C03654=1154.886,184.400,-60.410,-178.214,7.081,148.800
C03655=1154.890,184.131,-60.386,-178.217,7.080,148.800
C03656=1154.895,183.861,-60.360,-178.220,7.077,148.801
C03657=1154.900,183.591,-60.335,-178.223,7.075,148.801
C03658=1154.905,183.322,-60.310,-178.226,7.073,148.801
C03659=1154.909,183.073,-60.287,-178.229,7.070,148.801
C03660=1154.915,182.824,-60.264,-178.231,7.068,148.802
C03661=1154.919,182.576,-60.241,-178.234,7.066,148.802
C03662=1154.924,182.326,-60.218,-178.237,7.063,148.802
C03663=1154.928,182.077,-60.195,-178.240,7.062,148.803
C03664=1154.932,181.828,-60.172,-178.242,7.060,148.803
C03665=1154.938,181.580,-60.149,-178.245,7.057,148.803
C03666=1154.942,181.331,-60.126,-178.248,7.055,148.804
C03667=1154.946,181.082,-60.103,-178.251,7.053,148.804
C03668=1154.951,180.832,-60.080,-178.254,7.051,148.804
C03669=1154.956,180.583,-60.057,-178.256,7.049,148.804
C03670=1154.961,180.335,-60.035,-178.259,7.046,148.805
C03671=1154.965,180.086,-60.011,-178.262,7.045,148.805
C03672=1154.970,179.837,-59.989,-178.264,7.043,148.805
C03673=1154.974,179.588,-59.966,-178.267,7.040,148.806
C03674=1154.979,179.339,-59.943,-178.270,7.038,148.806
C03675=1154.984,179.091,-59.920,-178.272,7.036,148.806
C03676=1154.989,178.841,-59.898,-178.276,7.034,148.806
C03677=1154.993,178.593,-59.875,-178.278,7.032,148.807
C03678=1154.997,178.343,-59.851,-178.281,7.030,148.807
C03679=1155.002,178.095,-59.830,-178.284,7.027,148.807
C03680=1155.007,177.846,-59.806,-178.286,7.025,148.808
C03681=1155.012,177.596,-59.784,-178.289,7.024,148.808
C03682=1155.016,177.348,-59.761,-178.292,7.021,148.808
C03683=1155.021,177.099,-59.738,-178.295,7.019,148.808
C03684=1155.025,176.850,-59.716,-178.297,7.017,148.809
C03685=1155.030,176.601,-59.693,-178.301,7.015,148.809
C03686=1155.035,176.352,-59.671,-178.303,7.013,148.809
C03687=1155.040,176.103,-59.648,-178.306,7.011,148.810
C03688=1155.044,175.854,-59.625,-178.309,7.008,148.810
C03689=1155.048,175.606,-59.603,-178.311,7.007,148.810
C03690=1155.053,175.357,-59.580,-178.314,7.004,148.811
C03691=1155.057,175.107,-59.558,-178.317,7.002,148.811
C03692=1155.063,174.859,-59.535,-178.320,7.000,148.811
C03693=1155.067,174.610,-59.513,-178.322,6.998,148.812
C03694=1155.072,174.361,-59.489,-178.325,6.996,148.812
C03695=1155.077,174.112,-59.468,-178.328,6.994,148.812
C03696=1155.082,173.862,-59.445,-178.331,6.992,148.812
C03697=1155.086,173.614,-59.422,-178.334,6.989,148.813
C03698=1155.090,173.365,-59.401,-178.336,6.987,148.813
C03699=1155.095,173.116,-59.377,-178.339,6.986,148.813
C03700=1155.099,172.867,-59.355,-178.341,6.984,148.814
C03701=1155.104,172.619,-59.333,-178.345,6.981,148.814
C03702=1155.109,172.369,-59.310,-178.347,6.979,148.814
C03703=1155.114,172.120,-59.288,-178.350,6.977,148.815
C03704=1155.118,171.871,-59.265,-178.353,6.975,148.815
C03705=1155.123,171.622,-59.243,-178.356,6.973,148.815
C03706=1155.128,171.373,-59.221,-178.358,6.971,148.815
C03707=1155.132,171.124,-59.198,-178.361,6.969,148.816
C03708=1155.137,170.876,-59.176,-178.364,6.967,148.816
C03709=1155.141,170.626,-59.154,-178.366,6.965,148.817
C03710=1155.145,170.378,-59.131,-178.369,6.963,148.817
C03711=1155.151,170.129,-59.109,-178.372,6.960,148.817
C03712=1155.155,169.879,-59.087,-178.375,6.959,148.817
C03713=1155.160,169.631,-59.065,-178.377,6.957,148.818
C03714=1155.165,169.382,-59.042,-178.380,6.955,148.818
C03715=1155.170,169.133,-59.020,-178.383,6.953,148.818
C03716=1155.174,168.884,-58.998,-178.386,6.951,148.819
C03717=1155.179,168.635,-58.977,-178.388,6.949,148.819
C03718=1155.184,168.385,-58.954,-178.392,6.946,148.819
C03719=1155.188,168.137,-58.932,-178.394,6.945,148.820
C03720=1155.193,167.888,-58.910,-178.397,6.943,148.820
C03721=1155.197,167.639,-58.888,-178.399,6.941,148.820
C03722=1155.203,167.390,-58.865,-178.402,6.938,148.821
C03723=1155.207,167.140,-58.843,-178.405,6.936,148.821
C03724=1155.212,166.892,-58.822,-178.408,6.935,148.821
C03725=1155.216,166.642,-58.799,-178.411,6.933,148.822
C03726=1155.221,166.394,-58.778,-178.413,6.930,148.822
C03727=1155.225,166.145,-58.755,-178.416,6.928,148.822
C03728=1155.230,165.896,-58.733,-178.419,6.927,148.823
C03729=1155.235,165.647,-58.711,-178.421,6.925,148.823
C03730=1155.240,165.398,-58.689,-178.425,6.922,148.823
C03731=1155.244,165.149,-58.667,-178.427,6.920,148.823
C03732=1155.249,164.900,-58.645,-178.430,6.918,148.824
C03733=1155.254,164.651,-58.624,-178.432,6.917,148.824
C03734=1155.258,164.402,-58.602,-178.436,6.914,148.825
C03735=1155.263,164.153,-58.580,-178.438,6.912,148.825
C03736=1155.268,163.904,-58.557,-178.441,6.911,148.825
C03737=1155.273,163.655,-58.536,-178.443,6.909,148.825
C03738=1155.277,163.406,-58.513,-178.446,6.906,148.826
C03739=1155.282,163.157,-58.492,-178.449,6.904,148.826
C03740=1155.286,162.908,-58.470,-178.452,6.903,148.827
C03741=1155.291,162.659,-58.448,-178.455,6.901,148.827
C03742=1155.296,162.410,-58.427,-178.457,6.899,148.827
C03743=1155.300,162.161,-58.405,-178.461,6.897,148.828
C03744=1155.305,161.912,-58.383,-178.463,6.894,148.828
C03745=1155.309,161.663,-58.361,-178.465,6.893,148.828
C03746=1155.314,161.414,-58.340,-178.468,6.891,148.829
C03747=1155.319,161.165,-58.318,-178.471,6.888,148.829
C03748=1155.323,160.916,-58.296,-178.474,6.887,148.829
C03749=1155.328,160.667,-58.274,-178.477,6.885,148.830
C03750=1155.333,160.417,-58.253,-178.480,6.883,148.830
C03751=1155.338,160.169,-58.231,-178.482,6.881,148.830
C03752=1155.343,159.920,-58.210,-178.485,6.879,148.831
C03753=1155.347,159.671,-58.187,-178.488,6.877,148.831
C03754=1155.352,159.421,-58.167,-178.490,6.875,148.831
C03755=1155.357,159.173,-58.145,-178.493,6.873,148.832
C03756=1155.361,158.924,-58.123,-178.496,6.872,148.832
C03757=1155.366,158.675,-58.101,-178.499,6.869,148.832
C03758=1155.371,158.426,-58.080,-178.501,6.867,148.833
C03759=1155.376,158.157,-58.057,-178.504,6.865,148.833
C03760=1155.381,157.888,-58.033,-178.508,6.863,148.834
C03761=1155.386,157.619,-58.011,-178.511,6.861,148.834
C03762=1155.391,157.350,-57.986,-178.514,6.859,148.834
C03763=1155.396,157.101,-57.966,-178.516,6.857,148.834
C03764=1155.400,156.852,-57.944,-178.519,6.855,148.835
C03765=1155.405,156.603,-57.922,-178.521,6.853,148.835
C03766=1155.410,156.354,-57.901,-178.524,6.851,148.836
C03767=1155.414,156.105,-57.879,-178.527,6.850,148.836
C03768=1155.419,155.855,-57.858,-178.530,6.847,148.836
C03769=1155.424,155.607,-57.837,-178.533,6.845,148.837
C03770=1155.428,155.358,-57.815,-178.536,6.844,148.837
C03771=1155.433,155.108,-57.794,-178.538,6.842,148.837
C03772=1155.438,154.860,-57.773,-178.541,6.840,148.838
C03773=1155.443,154.610,-57.752,-178.543,6.838,148.838
C03774=1155.447,154.361,-57.730,-178.546,6.836,148.838
C03775=1155.452,154.112,-57.709,-178.549,6.834,148.839
C03776=1155.456,153.863,-57.688,-178.552,6.832,148.839
C03777=1155.462,153.614,-57.667,-178.555,6.830,148.839
C03778=1155.466,153.365,-57.645,-178.557,6.829,148.840
C03779=1155.471,153.116,-57.624,-178.560,6.827,148.840
C03780=1155.475,152.867,-57.602,-178.563,6.824,148.841
C03781=1155.480,152.618,-57.582,-178.566,6.823,148.841
C03782=1155.485,152.369,-57.560,-178.569,6.821,148.841
C03783=1155.490,152.119,-57.538,-178.571,6.819,148.842
C03784=1155.494,151.871,-57.517,-178.574,6.817,148.842
C03785=1155.499,151.622,-57.496,-178.576,6.815,148.842
C03786=1155.504,151.373,-57.475,-178.579,6.814,148.843
C03787=1155.508,151.124,-57.454,-178.582,6.811,148.843
C03788=1155.513,150.874,-57.433,-178.585,6.809,148.843
C03789=1155.518,150.625,-57.412,-178.588,6.808,148.844
C03790=1155.522,150.377,-57.391,-178.590,6.806,148.844
C03791=1155.528,150.127,-57.370,-178.593,6.804,148.845
C03792=1155.533,149.878,-57.349,-178.596,6.803,148.845
C03793=1155.537,149.630,-57.328,-178.598,6.801,148.845
C03794=1155.541,149.380,-57.307,-178.601,6.799,148.846
C03795=1155.547,149.131,-57.286,-178.604,6.797,148.846
C03796=1155.551,148.882,-57.265,-178.607,6.795,148.846
C03797=1155.556,148.633,-57.244,-178.610,6.793,148.847
C03798=1155.561,148.384,-57.223,-178.613,6.791,148.847
C03799=1155.565,148.135,-57.202,-178.615,6.790,148.848
C03800=1155.570,147.886,-57.181,-178.618,6.788,148.848
C03801=1155.574,147.637,-57.160,-178.620,6.786,148.848
C03802=1155.579,147.387,-57.139,-178.623,6.784,148.849
C03803=1155.585,147.138,-57.118,-178.626,6.782,148.849
C03804=1155.589,146.890,-57.097,-178.629,6.780,148.849
C03805=1155.594,146.640,-57.076,-178.632,6.778,148.850
C03806=1155.598,146.391,-57.055,-178.634,6.776,148.850
C03807=1155.603,146.142,-57.035,-178.637,6.775,148.850
C03808=1155.608,145.893,-57.014,-178.640,6.773,148.851
C03809=1155.613,145.644,-56.993,-178.642,6.771,148.851
C03810=1155.618,145.395,-56.973,-178.645,6.769,148.852
C03811=1155.622,145.146,-56.951,-178.648,6.768,148.852
C03812=1155.626,144.897,-56.930,-178.651,6.766,148.852
C03813=1155.631,144.648,-56.909,-178.653,6.764,148.853
C03814=1155.636,144.399,-56.889,-178.657,6.762,148.853
C03815=1155.641,144.149,-56.868,-178.659,6.760,148.853
C03816=1155.645,143.900,-56.848,-178.662,6.758,148.854
C03817=1155.651,143.651,-56.827,-178.665,6.757,148.854
C03818=1155.655,143.402,-56.806,-178.667,6.755,148.855
C03819=1155.660,143.153,-56.785,-178.670,6.753,148.855
C03820=1155.665,142.904,-56.765,-178.673,6.751,148.855
C03821=1155.669,142.655,-56.745,-178.676,6.750,148.856
C03822=1155.674,142.406,-56.724,-178.678,6.748,148.856
C03823=1155.679,142.157,-56.703,-178.681,6.746,148.857
C03824=1155.684,141.908,-56.682,-178.684,6.745,148.857
C03825=1155.688,141.659,-56.662,-178.686,6.743,148.857
C03826=1155.694,141.409,-56.641,-178.689,6.741,148.858
C03827=1155.698,141.160,-56.621,-178.692,6.739,148.858
C03828=1155.702,140.911,-56.600,-178.695,6.737,148.859
C03829=1155.708,140.662,-56.579,-178.698,6.735,148.859
C03830=1155.712,140.413,-56.559,-178.700,6.733,148.859
C03831=1155.716,140.164,-56.539,-178.703,6.732,148.860
C03832=1155.722,139.914,-56.518,-178.706,6.730,148.860
C03833=1155.726,139.665,-56.498,-178.709,6.728,148.860
C03834=1155.731,139.416,-56.478,-178.711,6.726,148.861
C03835=1155.736,139.167,-56.457,-178.714,6.725,148.861
C03836=1155.740,138.918,-56.436,-178.717,6.723,148.862
C03837=1155.745,138.669,-56.416,-178.719,6.721,148.862
C03838=1155.750,138.419,-56.396,-178.722,6.720,148.862
C03839=1155.755,138.171,-56.375,-178.725,6.718,148.863
C03840=1155.759,137.922,-56.355,-178.728,6.716,148.863
C03841=1155.764,137.672,-56.334,-178.730,6.714,148.864
C03842=1155.769,137.423,-56.314,-178.733,6.713,148.864
C03843=1155.774,137.174,-56.294,-178.736,6.711,148.864
C03844=1155.779,136.926,-56.274,-178.738,6.709,148.865
C03845=1155.784,136.676,-56.253,-178.741,6.708,148.865
C03846=1155.788,136.427,-56.233,-178.744,6.706,148.866
C03847=1155.793,136.178,-56.213,-178.747,6.704,148.866
C03848=1155.797,135.929,-56.193,-178.749,6.702,148.866
C03849=1155.803,135.680,-56.172,-178.752,6.701,148.867
C03850=1155.807,135.430,-56.152,-178.755,6.699,148.867
C03851=1155.812,135.181,-56.132,-178.757,6.697,148.867
C03852=1155.816,134.932,-56.111,-178.761,6.695,148.868
C03853=1155.822,134.683,-56.092,-178.764,6.693,148.868
C03854=1155.827,134.434,-56.071,-178.767,6.692,148.869
C03855=1155.831,134.185,-56.051,-178.769,6.690,148.869
C03856=1155.836,133.935,-56.031,-178.772,6.688,148.870
C03857=1155.840,133.686,-56.010,-178.775,6.686,148.870
C03858=1155.845,133.437,-55.991,-178.777,6.685,148.870
C03859=1155.849,133.188,-55.970,-178.780,6.683,148.871
C03860=1155.855,132.939,-55.951,-178.783,6.681,148.871
C03861=1155.860,132.690,-55.930,-178.786,6.680,148.872
C03862=1155.864,132.441,-55.910,-178.788,6.678,148.872
C03863=1155.869,132.172,-55.889,-178.791,6.676,148.872
C03864=1155.875,131.903,-55.867,-178.794,6.674,148.873
C03865=1155.880,131.635,-55.845,-178.797,6.673,148.873
C03866=1155.885,131.366,-55.824,-178.800,6.671,148.874
C03867=1155.890,131.117,-55.804,-178.802,6.670,148.874
C03868=1155.894,130.868,-55.784,-178.805,6.668,148.875
C03869=1155.900,130.619,-55.764,-178.808,6.666,148.875
C03870=1155.904,130.370,-55.744,-178.810,6.664,148.875
C03871=1155.909,130.120,-55.724,-178.813,6.663,148.876
C03872=1155.913,129.871,-55.704,-178.816,6.661,148.876
C03873=1155.919,129.623,-55.685,-178.819,6.659,148.877
C03874=1155.923,129.373,-55.665,-178.821,6.658,148.877
C03875=1155.928,129.124,-55.645,-178.824,6.656,148.878
C03876=1155.933,128.874,-55.625,-178.827,6.655,148.878
C03877=1155.938,128.626,-55.605,-178.830,6.653,148.878
C03878=1155.942,128.377,-55.585,-178.833,6.651,148.879
C03879=1155.947,128.127,-55.566,-178.835,6.649,148.879
C03880=1155.952,127.878,-55.545,-178.838,6.648,148.880
C03881=1155.957,127.629,-55.526,-178.841,6.646,148.880
C03882=1155.962,127.380,-55.506,-178.843,6.644,148.880
C03883=1155.966,127.131,-55.486,-178.846,6.643,148.881
C03884=1155.971,126.881,-55.466,-178.849,6.641,148.881
C03885=1155.976,126.632,-55.447,-178.852,6.639,148.882
C03886=1155.981,126.383,-55.427,-178.855,6.638,148.882
C03887=1155.985,126.134,-55.407,-178.858,6.636,148.883
C03888=1155.991,125.885,-55.388,-178.860,6.634,148.883
C03889=1155.996,125.635,-55.368,-178.863,6.633,148.883
C03890=1155.999,125.387,-55.348,-178.866,6.631,148.884
C03891=1156.004,125.137,-55.329,-178.868,6.629,148.884
C03892=1156.009,124.888,-55.309,-178.871,6.627,148.885
C03893=1156.014,124.639,-55.290,-178.874,6.626,148.885
C03894=1156.019,124.389,-55.270,-178.876,6.625,148.885
C03895=1156.024,124.141,-55.250,-178.879,6.623,148.886
C03896=1156.029,123.891,-55.230,-178.882,6.622,148.886
C03897=1156.033,123.642,-55.211,-178.885,6.620,148.887
C03898=1156.038,123.393,-55.192,-178.887,6.618,148.887
C03899=1156.043,123.144,-55.172,-178.890,6.617,148.888
C03900=1156.047,122.894,-55.153,-178.893,6.615,148.888
C03901=1156.053,122.645,-55.133,-178.895,6.613,148.888
C03902=1156.057,122.396,-55.114,-178.898,6.612,148.889
C03903=1156.063,122.147,-55.094,-178.901,6.610,148.889
C03904=1156.067,121.898,-55.075,-178.904,6.608,148.890
C03905=1156.071,121.649,-55.055,-178.907,6.607,148.890
C03906=1156.077,121.400,-55.036,-178.909,6.605,148.891
C03907=1156.081,121.150,-55.016,-178.912,6.603,148.891
C03908=1156.086,120.901,-54.996,-178.914,6.602,148.891
C03909=1156.091,120.652,-54.978,-178.917,6.601,148.892
C03910=1156.095,120.402,-54.958,-178.920,6.599,148.892
C03911=1156.101,120.154,-54.939,-178.922,6.597,148.893
C03912=1156.106,119.904,-54.919,-178.926,6.596,148.893
C03913=1156.110,119.655,-54.900,-178.928,6.594,148.894
C03914=1156.115,119.406,-54.881,-178.931,6.593,148.894
C03915=1156.120,119.156,-54.861,-178.934,6.591,148.894
C03916=1156.125,118.907,-54.842,-178.937,6.589,148.895
C03917=1156.129,118.658,-54.823,-178.939,6.587,148.895
C03918=1156.134,118.409,-54.803,-178.941,6.587,148.896
C03919=1156.139,118.160,-54.784,-178.945,6.585,148.896
C03920=1156.144,117.911,-54.766,-178.947,6.583,148.897
C03921=1156.149,117.661,-54.746,-178.950,6.582,148.897
C03922=1156.154,117.412,-54.727,-178.953,6.580,148.897
C03923=1156.158,117.163,-54.708,-178.955,6.578,148.898
C03924=1156.163,116.913,-54.688,-178.958,6.577,148.898
C03925=1156.168,116.664,-54.669,-178.961,6.575,148.899
C03926=1156.172,116.415,-54.650,-178.964,6.574,148.899
C03927=1156.178,116.166,-54.630,-178.966,6.573,148.900
C03928=1156.183,115.916,-54.611,-178.969,6.571,148.900
C03929=1156.187,115.668,-54.593,-178.972,6.569,148.901
C03930=1156.192,115.418,-54.573,-178.974,6.568,148.901
C03931=1156.197,115.169,-54.554,-178.977,6.566,148.901
C03932=1156.201,114.920,-54.535,-178.980,6.565,148.902
C03933=1156.207,114.670,-54.516,-178.983,6.563,148.902
C03934=1156.211,114.421,-54.497,-178.986,6.561,148.903
C03935=1156.216,114.172,-54.478,-178.988,6.560,148.903
C03936=1156.221,113.924,-54.459,-178.991,6.558,148.904
C03937=1156.226,113.674,-54.440,-178.993,6.557,148.904
C03938=1156.231,113.425,-54.421,-178.997,6.555,148.905
C03939=1156.235,113.175,-54.402,-178.999,6.554,148.905
C03940=1156.241,112.926,-54.383,-179.002,6.552,148.905
C03941=1156.245,112.677,-54.364,-179.005,6.550,148.906
C03942=1156.250,112.428,-54.345,-179.007,6.549,148.906
C03943=1156.255,112.178,-54.327,-179.010,6.548,148.907
C03944=1156.260,111.929,-54.307,-179.013,6.546,148.907
C03945=1156.265,111.681,-54.289,-179.015,6.545,148.908
C03946=1156.270,111.430,-54.270,-179.018,6.543,148.908
C03947=1156.274,111.182,-54.251,-179.021,6.541,148.909
C03948=1156.279,110.932,-54.232,-179.024,6.540,148.909
C03949=1156.284,110.683,-54.213,-179.026,6.539,148.910
C03950=1156.289,110.433,-54.194,-179.029,6.537,148.910
C03951=1156.293,110.184,-54.176,-179.032,6.536,148.910
C03952=1156.299,109.935,-54.156,-179.034,6.534,148.911
C03953=1156.303,109.686,-54.138,-179.037,6.532,148.911
C03954=1156.308,109.437,-54.119,-179.040,6.531,148.912
C03955=1156.313,109.188,-54.101,-179.042,6.530,148.912
C03956=1156.317,108.938,-54.082,-179.045,6.528,148.913
C03957=1156.323,108.689,-54.063,-179.048,6.527,148.913
C03958=1156.327,108.440,-54.044,-179.051,6.525,148.913
C03959=1156.333,108.190,-54.026,-179.054,6.524,148.914
C03960=1156.337,107.941,-54.007,-179.056,6.523,148.915
C03961=1156.342,107.691,-53.988,-179.059,6.521,148.915
C03962=1156.347,107.443,-53.969,-179.061,6.519,148.915
C03963=1156.352,107.194,-53.951,-179.064,6.518,148.916
C03964=1156.357,106.944,-53.932,-179.067,6.516,148.916
C03965=1156.362,106.695,-53.914,-179.070,6.515,148.917
C03966=1156.366,106.446,-53.895,-179.072,6.514,148.917
C03967=1156.371,106.177,-53.875,-179.075,6.512,148.918
C03968=1156.376,105.909,-53.855,-179.078,6.511,148.918
C03969=1156.382,105.641,-53.834,-179.081,6.509,148.919
C03970=1156.387,105.373,-53.815,-179.084,6.508,148.919
C03971=1156.392,105.122,-53.796,-179.087,6.506,148.920
C03972=1156.397,104.874,-53.777,-179.090,6.504,148.920
C03973=1156.402,104.625,-53.759,-179.092,6.502,148.921
C03974=1156.407,104.374,-53.740,-179.095,6.501,148.921
C03975=1156.412,104.125,-53.722,-179.098,6.500,148.922
C03976=1156.416,103.877,-53.704,-179.100,6.499,148.922
C03977=1156.421,103.628,-53.686,-179.103,6.497,148.922
C03978=1156.426,103.377,-53.667,-179.106,6.495,148.923
C03979=1156.431,103.129,-53.648,-179.109,6.494,148.923
C03980=1156.436,102.880,-53.630,-179.111,6.493,148.924
C03981=1156.441,102.630,-53.612,-179.114,6.491,148.924
C03982=1156.446,102.380,-53.593,-179.117,6.490,148.925
C03983=1156.450,102.132,-53.575,-179.120,6.488,148.925
C03984=1156.455,101.882,-53.557,-179.122,6.487,148.926
C03985=1156.460,101.633,-53.539,-179.125,6.486,148.926
C03986=1156.465,101.383,-53.520,-179.127,6.484,148.927
C03987=1156.470,101.135,-53.501,-179.131,6.483,148.927
C03988=1156.475,100.885,-53.483,-179.133,6.481,148.928
C03989=1156.480,100.636,-53.465,-179.135,6.480,148.928
C03990=1156.484,100.386,-53.447,-179.138,6.478,148.928
C03991=1156.489,100.137,-53.428,-179.141,6.477,148.929
C03992=1156.494,99.888,-53.410,-179.144,6.475,148.929
C03993=1156.499,99.639,-53.392,-179.146,6.474,148.930
C03994=1156.504,99.390,-53.373,-179.149,6.473,148.930
C03995=1156.508,99.140,-53.355,-179.152,6.471,148.931
C03996=1156.513,98.891,-53.337,-179.155,6.470,148.931
C03997=1156.518,98.642,-53.319,-179.157,6.469,148.932
C03998=1156.524,98.392,-53.301,-179.160,6.467,148.932
C03999=1156.529,98.143,-53.283,-179.163,6.466,148.933
C04000=1156.534,97.894,-53.265,-179.166,6.464,148.933
C04001=1156.538,97.644,-53.246,-179.168,6.463,148.934
C04002=1156.543,97.395,-53.228,-179.171,6.461,148.934
C04003=1156.548,97.146,-53.210,-179.174,6.460,148.935
C04004=1156.553,96.896,-53.192,-179.176,6.458,148.935
C04005=1156.557,96.647,-53.174,-179.179,6.458,148.936
C04006=1156.562,96.398,-53.156,-179.181,6.456,148.936
C04007=1156.567,96.148,-53.138,-179.185,6.455,148.937
C04008=1156.572,95.899,-53.120,-179.187,6.453,148.937
C04009=1156.577,95.650,-53.102,-179.189,6.452,148.937
C04010=1156.581,95.401,-53.084,-179.192,6.450,148.938
C04011=1156.586,95.152,-53.066,-179.195,6.449,148.939
C04012=1156.591,94.902,-53.048,-179.197,6.448,148.939
C04013=1156.597,94.653,-53.029,-179.200,6.446,148.939
C04014=1156.602,94.404,-53.012,-179.203,6.445,148.940
C04015=1156.607,94.155,-52.994,-179.206,6.443,148.940
C04016=1156.611,93.905,-52.975,-179.208,6.442,148.941
C04017=1156.616,93.655,-52.957,-179.211,6.441,148.941
C04018=1156.621,93.406,-52.940,-179.214,6.439,148.942
C04019=1156.625,93.157,-52.923,-179.216,6.439,148.942
C04020=1156.630,92.908,-52.905,-179.219,6.437,148.943
C04021=1156.635,92.658,-52.887,-179.222,6.436,148.943
C04022=1156.640,92.409,-52.869,-179.225,6.434,148.944
C04023=1156.645,92.160,-52.851,-179.227,6.433,148.944
C04024=1156.650,91.910,-52.833,-179.230,6.431,148.945
C04025=1156.655,91.661,-52.815,-179.233,6.430,148.945
C04026=1156.660,91.412,-52.797,-179.235,6.429,148.946
C04027=1156.665,91.163,-52.779,-179.238,6.427,148.946
C04028=1156.670,90.914,-52.761,-179.241,6.426,148.947
C04029=1156.675,90.664,-52.744,-179.244,6.424,148.947
C04030=1156.680,90.415,-52.726,-179.246,6.423,148.948
C04031=1156.685,90.165,-52.708,-179.249,6.422,148.948
C04032=1156.689,89.917,-52.691,-179.252,6.420,148.949
C04033=1156.694,89.666,-52.673,-179.254,6.420,148.949
C04034=1156.699,89.417,-52.655,-179.257,6.418,148.950
C04035=1156.704,89.168,-52.637,-179.260,6.417,148.950
C04036=1156.709,88.918,-52.620,-179.262,6.416,148.951
C04037=1156.714,88.669,-52.602,-179.265,6.414,148.951
C04038=1156.719,88.420,-52.584,-179.268,6.413,148.952
C04039=1156.723,88.170,-52.567,-179.270,6.412,148.952
C04040=1156.728,87.921,-52.549,-179.273,6.410,148.953
C04041=1156.733,87.672,-52.532,-179.276,6.408,148.953
C04042=1156.739,87.423,-52.515,-179.278,6.408,148.954
C04043=1156.744,87.174,-52.497,-179.281,6.406,148.954
C04044=1156.749,86.924,-52.479,-179.284,6.405,148.954
C04045=1156.753,86.675,-52.462,-179.287,6.404,148.955
C04046=1156.758,86.426,-52.444,-179.289,6.402,148.955
C04047=1156.763,86.176,-52.427,-179.292,6.401,148.956
C04048=1156.768,85.927,-52.409,-179.295,6.400,148.957
C04049=1156.773,85.677,-52.392,-179.297,6.398,148.957
C04050=1156.777,85.428,-52.374,-179.300,6.397,148.957
C04051=1156.783,85.178,-52.357,-179.303,6.396,148.958
C04052=1156.788,84.929,-52.339,-179.305,6.395,148.958
C04053=1156.792,84.680,-52.321,-179.308,6.393,148.959
C04054=1156.797,84.430,-52.304,-179.311,6.392,148.960
C04055=1156.802,84.181,-52.286,-179.314,6.391,148.960
C04056=1156.807,83.931,-52.269,-179.316,6.389,148.960
C04057=1156.812,83.682,-52.252,-179.319,6.388,148.961
C04058=1156.816,83.433,-52.234,-179.322,6.387,148.961
C04059=1156.822,83.184,-52.217,-179.324,6.385,148.962
C04060=1156.826,82.935,-52.200,-179.327,6.385,148.963
C04061=1156.832,82.685,-52.183,-179.330,6.383,148.963
C04062=1156.837,82.436,-52.165,-179.332,6.381,148.963
C04063=1156.841,82.186,-52.148,-179.335,6.380,148.964
C04064=1156.846,81.937,-52.130,-179.338,6.379,148.964
C04065=1156.851,81.687,-52.113,-179.340,6.378,148.965
C04066=1156.856,81.438,-52.096,-179.343,6.376,148.965
C04067=1156.861,81.189,-52.078,-179.346,6.375,148.966
C04068=1156.866,80.940,-52.061,-179.348,6.374,148.966
C04069=1156.871,80.690,-52.045,-179.351,6.373,148.967
C04070=1156.876,80.441,-52.027,-179.354,6.371,148.967
C04071=1156.881,80.172,-52.008,-179.356,6.370,148.968
C04072=1156.886,79.904,-51.990,-179.359,6.369,148.969
C04073=1156.892,79.635,-51.971,-179.362,6.367,148.969
C04074=1156.897,79.367,-51.953,-179.365,6.366,148.970
C04075=1156.902,79.118,-51.936,-179.367,6.365,148.970
C04076=1156.907,78.869,-51.918,-179.371,6.364,148.971
C04077=1156.912,78.619,-51.902,-179.373,6.362,148.971
C04078=1156.917,78.370,-51.884,-179.376,6.361,148.972
C04079=1156.921,78.120,-51.867,-179.379,6.360,148.972
C04080=1156.927,77.871,-51.850,-179.382,6.358,148.973
C04081=1156.931,77.622,-51.834,-179.384,6.358,148.973
C04082=1156.936,77.373,-51.816,-179.387,6.356,148.974
C04083=1156.942,77.123,-51.798,-179.389,6.355,148.974
C04084=1156.946,76.873,-51.782,-179.392,6.354,148.975
C04085=1156.952,76.624,-51.765,-179.395,6.352,148.975
C04086=1156.956,76.375,-51.748,-179.397,6.351,148.976
C04087=1156.961,76.126,-51.730,-179.400,6.350,148.976
C04088=1156.966,75.876,-51.713,-179.402,6.349,148.977
C04089=1156.972,75.627,-51.697,-179.405,6.348,148.977
C04090=1156.976,75.378,-51.680,-179.408,6.347,148.978
C04091=1156.980,75.128,-51.663,-179.411,6.345,148.978
C04092=1156.986,74.878,-51.646,-179.413,6.344,148.979
C04093=1156.990,74.629,-51.629,-179.416,6.343,148.979
C04094=1156.996,74.380,-51.612,-179.419,6.342,148.980
C04095=1157.000,74.131,-51.595,-179.421,6.341,148.980
C04096=1157.005,73.881,-51.578,-179.424,6.339,148.981
C04097=1157.010,73.632,-51.561,-179.427,6.338,148.981
C04098=1157.016,73.382,-51.544,-179.429,6.337,148.982
C04099=1157.020,73.133,-51.528,-179.432,6.336,148.982
C04100=1157.025,72.883,-51.511,-179.434,6.335,148.983
C04101=1157.030,72.634,-51.494,-179.438,6.333,148.983
C04102=1157.035,72.385,-51.477,-179.440,6.332,148.984
C04103=1157.040,72.135,-51.460,-179.442,6.331,148.984
C04104=1157.045,71.886,-51.444,-179.446,6.329,148.985
C04105=1157.050,71.637,-51.427,-179.448,6.329,148.985
C04106=1157.055,71.387,-51.410,-179.451,6.327,148.986
C04107=1157.060,71.138,-51.393,-179.453,6.326,148.987
C04108=1157.064,70.889,-51.377,-179.456,6.325,148.987
C04109=1157.070,70.639,-51.360,-179.459,6.324,148.988
C04110=1157.075,70.390,-51.343,-179.461,6.323,148.988
C04111=1157.079,70.141,-51.327,-179.463,6.322,148.988
C04112=1157.084,69.891,-51.309,-179.467,6.320,148.989
C04113=1157.090,69.642,-51.293,-179.469,6.319,148.990
C04114=1157.094,69.392,-51.277,-179.472,6.318,148.990
C04115=1157.100,69.142,-51.260,-179.475,6.317,148.991
C04116=1157.105,68.893,-51.243,-179.477,6.316,148.991
C04117=1157.109,68.644,-51.227,-179.480,6.314,148.992
C04118=1157.114,68.394,-51.210,-179.482,6.314,148.992
C04119=1157.119,68.145,-51.193,-179.485,6.312,148.993
C04120=1157.124,67.896,-51.177,-179.488,6.311,148.993
C04121=1157.128,67.646,-51.160,-179.490,6.310,148.994
C04122=1157.135,67.397,-51.144,-179.493,6.309,148.994
C04123=1157.139,67.147,-51.127,-179.496,6.308,148.995
C04124=1157.144,66.898,-51.111,-179.498,6.307,148.995
C04125=1157.149,66.649,-51.094,-179.501,6.305,148.996
C04126=1157.154,66.399,-51.077,-179.504,6.304,148.996
C04127=1157.159,66.150,-51.061,-179.507,6.303,148.997
C04128=1157.164,65.900,-51.045,-179.509,6.301,148.997
C04129=1157.169,65.652,-51.028,-179.511,6.301,148.998
C04130=1157.173,65.402,-51.012,-179.515,6.299,148.999
C04131=1157.179,65.152,-50.995,-179.517,6.298,148.999
C04132=1157.184,64.903,-50.979,-179.520,6.297,149.000
C04133=1157.188,64.653,-50.962,-179.522,6.296,149.000
C04134=1157.193,64.405,-50.946,-179.525,6.295,149.000
C04135=1157.198,64.154,-50.930,-179.528,6.294,149.001
C04136=1157.203,63.906,-50.913,-179.530,6.292,149.002
C04137=1157.208,63.656,-50.896,-179.533,6.292,149.002
C04138=1157.214,63.406,-50.881,-179.536,6.290,149.003
C04139=1157.218,63.157,-50.864,-179.538,6.289,149.003
C04140=1157.223,62.908,-50.847,-179.541,6.288,149.004
C04141=1157.228,62.658,-50.832,-179.543,6.287,149.004
C04142=1157.233,62.409,-50.815,-179.546,6.286,149.005
C04143=1157.238,62.159,-50.799,-179.549,6.285,149.005
C04144=1157.243,61.909,-50.782,-179.551,6.283,149.006
C04145=1157.248,61.661,-50.766,-179.554,6.283,149.006
C04146=1157.253,61.411,-50.750,-179.557,6.281,149.007
C04147=1157.258,61.162,-50.734,-179.559,6.281,149.008
C04148=1157.263,60.912,-50.718,-179.562,6.279,149.008
C04149=1157.268,60.663,-50.701,-179.564,6.278,149.008
C04150=1157.273,60.413,-50.685,-179.567,6.277,149.009
C04151=1157.278,60.164,-50.669,-179.570,6.276,149.009
C04152=1157.282,59.915,-50.652,-179.573,6.275,149.010
C04153=1157.288,59.665,-50.637,-179.575,6.274,149.011
C04154=1157.292,59.416,-50.620,-179.578,6.273,149.011
C04155=1157.298,59.166,-50.605,-179.580,6.272,149.012
C04156=1157.302,58.917,-50.588,-179.583,6.270,149.012
C04157=1157.308,58.667,-50.572,-179.586,6.270,149.013
C04158=1157.313,58.419,-50.556,-179.588,6.268,149.013
C04159=1157.317,58.168,-50.540,-179.591,6.267,149.014
C04160=1157.322,57.920,-50.524,-179.593,6.267,149.014
C04161=1157.327,57.670,-50.508,-179.596,6.265,149.015
C04162=1157.332,57.421,-50.492,-179.599,6.264,149.015
C04163=1157.337,57.171,-50.476,-179.601,6.263,149.016
C04164=1157.343,56.921,-50.460,-179.604,6.262,149.017
C04165=1157.347,56.672,-50.443,-179.607,6.261,149.017
C04166=1157.352,56.422,-50.428,-179.609,6.260,149.018
C04167=1157.357,56.174,-50.411,-179.612,6.258,149.018
C04168=1157.362,55.923,-50.395,-179.614,6.258,149.019
C04169=1157.368,55.674,-50.380,-179.618,6.256,149.019
C04170=1157.372,55.425,-50.363,-179.620,6.255,149.020
C04171=1157.378,55.175,-50.348,-179.623,6.254,149.020
C04172=1157.383,54.926,-50.332,-179.625,6.253,149.021
C04173=1157.387,54.676,-50.315,-179.628,6.253,149.021
C04174=1157.393,54.427,-50.300,-179.630,6.251,149.022
C04175=1157.398,54.158,-50.283,-179.634,6.250,149.022
C04176=1157.403,53.889,-50.265,-179.636,6.249,149.023
C04177=1157.409,53.621,-50.248,-179.639,6.248,149.024
C04178=1157.414,53.352,-50.231,-179.642,6.247,149.024
C04179=1157.420,53.103,-50.216,-179.644,6.246,149.025
C04180=1157.424,52.854,-50.200,-179.647,6.245,149.025
C04181=1157.429,52.604,-50.184,-179.650,6.243,149.026
C04182=1157.434,52.355,-50.169,-179.652,6.243,149.026
C04183=1157.439,52.105,-50.153,-179.655,6.241,149.027
C04184=1157.444,51.856,-50.136,-179.657,6.240,149.027
C04185=1157.450,51.607,-50.121,-179.660,6.240,149.028
C04186=1157.454,51.357,-50.105,-179.663,6.238,149.028
C04187=1157.459,51.107,-50.090,-179.665,6.237,149.029
C04188=1157.464,50.859,-50.073,-179.668,6.236,149.030
C04189=1157.469,50.609,-50.057,-179.670,6.235,149.030
C04190=1157.474,50.359,-50.042,-179.674,6.234,149.031
C04191=1157.479,50.110,-50.027,-179.676,6.233,149.031
C04192=1157.484,49.860,-50.011,-179.678,6.233,149.032
C04193=1157.489,49.611,-49.995,-179.681,6.231,149.032
C04194=1157.494,49.361,-49.980,-179.684,6.230,149.033
C04195=1157.499,49.112,-49.963,-179.686,6.229,149.033
C04196=1157.504,48.863,-49.948,-179.689,6.228,149.034
C04197=1157.509,48.613,-49.933,-179.691,6.227,149.034
C04198=1157.514,48.364,-49.917,-179.694,6.226,149.035
C04199=1157.519,48.114,-49.901,-179.697,6.225,149.036
C04200=1157.524,47.865,-49.886,-179.699,6.224,149.036
C04201=1157.529,47.615,-49.870,-179.702,6.223,149.037
C04202=1157.534,47.365,-49.854,-179.704,6.222,149.037
C04203=1157.539,47.116,-49.839,-179.707,6.221,149.038
C04204=1157.544,46.867,-49.824,-179.710,6.220,149.038
C04205=1157.549,46.617,-49.808,-179.713,6.219,149.039
C04206=1157.554,46.367,-49.792,-179.715,6.218,149.039
C04207=1157.559,46.118,-49.777,-179.717,6.217,149.040
C04208=1157.564,45.869,-49.762,-179.720,6.216,149.040
C04209=1157.570,45.619,-49.746,-179.723,6.215,149.041
C04210=1157.574,45.370,-49.731,-179.726,6.214,149.042
C04211=1157.579,45.120,-49.715,-179.728,6.213,149.042
C04212=1157.584,44.871,-49.700,-179.731,6.212,149.043
C04213=1157.589,44.621,-49.685,-179.733,6.211,149.043
C04214=1157.594,44.372,-49.669,-179.736,6.210,149.044
C04215=1157.599,44.122,-49.653,-179.739,6.209,149.044
C04216=1157.604,43.873,-49.638,-179.741,6.208,149.045
C04217=1157.609,43.623,-49.622,-179.744,6.207,149.045
C04218=1157.614,43.374,-49.607,-179.747,6.206,149.046
C04219=1157.619,43.125,-49.592,-179.749,6.205,149.047
C04220=1157.624,42.875,-49.576,-179.751,6.204,149.047
C04221=1157.629,42.626,-49.561,-179.754,6.203,149.048
C04222=1157.634,42.376,-49.546,-179.756,6.202,149.048
C04223=1157.639,42.127,-49.531,-179.759,6.202,149.049
C04224=1157.644,41.877,-49.516,-179.762,6.200,149.049
C04225=1157.650,41.628,-49.500,-179.764,6.200,149.050
C04226=1157.654,41.378,-49.485,-179.767,6.198,149.050
C04227=1157.659,41.129,-49.469,-179.770,6.197,149.051
C04228=1157.664,40.880,-49.454,-179.772,6.197,149.051
C04229=1157.670,40.630,-49.439,-179.775,6.195,149.052
C04230=1157.674,40.380,-49.424,-179.777,6.194,149.053
C04231=1157.680,40.131,-49.409,-179.780,6.194,149.053
C04232=1157.685,39.882,-49.393,-179.783,6.192,149.054
C04233=1157.689,39.631,-49.378,-179.785,6.192,149.054
C04234=1157.695,39.382,-49.363,-179.788,6.191,149.055
C04235=1157.699,39.133,-49.348,-179.791,6.190,149.055
C04236=1157.705,38.883,-49.332,-179.793,6.189,149.056
C04237=1157.710,38.634,-49.318,-179.795,6.188,149.056
C04238=1157.715,38.384,-49.302,-179.798,6.187,149.057
C04239=1157.720,38.135,-49.287,-179.801,6.186,149.057
C04240=1157.725,37.886,-49.272,-179.803,6.185,149.058
C04241=1157.730,37.636,-49.257,-179.806,6.184,149.059
C04242=1157.736,37.387,-49.242,-179.809,6.183,149.059
C04243=1157.740,37.137,-49.226,-179.811,6.182,149.060
C04244=1157.745,36.887,-49.212,-179.814,6.181,149.060
C04245=1157.750,36.638,-49.197,-179.816,6.180,149.061
C04246=1157.755,36.389,-49.182,-179.819,6.180,149.062
C04247=1157.760,36.139,-49.167,-179.822,6.178,149.062
C04248=1157.765,35.890,-49.152,-179.824,6.178,149.063
C04249=1157.770,35.640,-49.136,-179.826,6.177,149.063
C04250=1157.775,35.390,-49.122,-179.830,6.176,149.064
C04251=1157.780,35.141,-49.107,-179.832,6.175,149.064
C04252=1157.786,34.891,-49.092,-179.834,6.174,149.065
C04253=1157.790,34.642,-49.077,-179.837,6.173,149.065
C04254=1157.796,34.393,-49.061,-179.840,6.172,149.066
C04255=1157.801,34.143,-49.047,-179.842,6.171,149.066
C04256=1157.805,33.894,-49.032,-179.845,6.170,149.067
C04257=1157.811,33.644,-49.017,-179.847,6.169,149.068
C04258=1157.816,33.395,-49.002,-179.850,6.169,149.068
C04259=1157.821,33.145,-48.987,-179.853,6.167,149.069
C04260=1157.826,32.896,-48.972,-179.855,6.167,149.069
C04261=1157.831,32.646,-48.958,-179.858,6.166,149.070
C04262=1157.836,32.397,-48.943,-179.860,6.165,149.071
C04263=1157.841,32.147,-48.928,-179.863,6.164,149.071
C04264=1157.846,31.898,-48.913,-179.866,6.163,149.072
C04265=1157.852,31.648,-48.898,-179.868,6.162,149.072
C04266=1157.856,31.399,-48.883,-179.871,6.161,149.073
C04267=1157.861,31.149,-48.869,-179.873,6.160,149.073
C04268=1157.866,30.900,-48.854,-179.876,6.160,149.074
C04269=1157.872,30.650,-48.839,-179.879,6.158,149.074
C04270=1157.876,30.401,-48.824,-179.881,6.158,149.075
C04271=1157.881,30.151,-48.810,-179.883,6.157,149.075
C04272=1157.887,29.901,-48.795,-179.886,6.156,149.076
C04273=1157.891,29.652,-48.780,-179.889,6.155,149.077
C04274=1157.896,29.402,-48.766,-179.891,6.154,149.077
C04275=1157.901,29.153,-48.751,-179.894,6.153,149.078
C04276=1157.907,28.903,-48.736,-179.896,6.152,149.078
C04277=1157.912,28.653,-48.722,-179.899,6.151,149.079
C04278=1157.916,28.404,-48.707,-179.901,6.150,149.079
C04279=1157.922,28.136,-48.691,-179.904,6.149,149.080
C04280=1157.928,27.866,-48.675,-179.907,6.149,149.081
C04281=1157.933,27.597,-48.660,-179.910,6.148,149.081
C04282=1157.938,27.328,-48.644,-179.912,6.147,149.082
C04283=1157.944,27.078,-48.629,-179.915,6.146,149.082
C04284=1157.949,26.830,-48.615,-179.917,6.145,149.083
C04285=1157.954,26.580,-48.600,-179.921,6.144,149.084
C04286=1157.959,26.330,-48.586,-179.923,6.143,149.084
C04287=1157.963,26.081,-48.571,-179.925,6.143,149.085
C04288=1157.969,25.831,-48.556,-179.928,6.141,149.085
C04289=1157.974,25.582,-48.542,-179.931,6.141,149.086
C04290=1157.979,25.332,-48.528,-179.933,6.140,149.086
C04291=1157.984,25.083,-48.513,-179.936,6.139,149.087
C04292=1157.989,24.833,-48.498,-179.938,6.138,149.087
C04293=1157.994,24.584,-48.484,-179.941,6.137,149.088
C04294=1157.999,24.334,-48.470,-179.943,6.136,149.089
C04295=1158.005,24.084,-48.455,-179.946,6.136,149.089
C04296=1158.009,23.835,-48.440,-179.949,6.134,149.090
C04297=1158.014,23.586,-48.426,-179.951,6.134,149.090
C04298=1158.019,23.336,-48.412,-179.953,6.133,149.091
C04299=1158.024,23.086,-48.397,-179.956,6.132,149.092
C04300=1158.029,22.836,-48.383,-179.959,6.131,149.092
C04301=1158.035,22.588,-48.369,-179.961,6.130,149.093
C04302=1158.040,22.338,-48.354,-179.964,6.130,149.093
C04303=1158.044,22.089,-48.340,-179.966,6.129,149.094
C04304=1158.049,21.839,-48.326,-179.968,6.128,149.094
C04305=1158.054,21.589,-48.311,-179.972,6.127,149.095
C04306=1158.060,21.339,-48.297,-179.974,6.126,149.095
C04307=1158.066,21.090,-48.283,-179.976,6.126,149.096
C04308=1158.071,20.840,-48.268,-179.979,6.125,149.097
C04309=1158.076,20.591,-48.254,-179.982,6.124,149.097
C04310=1158.080,20.342,-48.239,-179.984,6.123,149.098
C04311=1158.085,20.092,-48.225,-179.987,6.122,149.098
C04312=1158.091,19.843,-48.211,-179.989,6.121,149.099
C04313=1158.096,19.593,-48.197,-179.992,6.120,149.100
C04314=1158.101,19.344,-48.182,-179.994,6.119,149.100
C04315=1158.106,19.094,-48.168,-179.997,6.119,149.101
C04316=1158.111,18.844,-48.154,-179.999,6.118,149.101
C04317=1158.116,18.595,-48.140,179.998,6.118,149.102
C04318=1158.121,18.345,-48.126,179.996,6.116,149.102
C04319=1158.126,18.096,-48.111,179.993,6.116,149.103
C04320=1158.131,17.846,-48.097,179.991,6.115,149.103
C04321=1158.136,17.597,-48.083,179.988,6.114,149.104
C04322=1158.141,17.347,-48.069,179.985,6.114,149.105
C04323=1158.146,17.098,-48.055,179.983,6.112,149.105
C04324=1158.151,16.848,-48.040,179.980,6.112,149.106
C04325=1158.157,16.599,-48.026,179.978,6.111,149.106
C04326=1158.161,16.349,-48.013,179.975,6.110,149.107
C04327=1158.166,16.099,-47.999,179.973,6.110,149.107
C04328=1158.171,15.849,-47.985,179.970,6.108,149.108
C04329=1158.177,15.600,-47.971,179.968,6.107,149.109
C04330=1158.182,15.351,-47.957,179.965,6.107,149.109
C04331=1158.187,15.101,-47.942,179.963,6.106,149.110
C04332=1158.192,14.852,-47.928,179.960,6.106,149.110
C04333=1158.197,14.602,-47.914,179.957,6.104,149.111
C04334=1158.202,14.353,-47.900,179.955,6.104,149.112
C04335=1158.207,14.103,-47.886,179.953,6.103,149.112
C04336=1158.212,13.853,-47.873,179.950,6.102,149.113
C04337=1158.217,13.604,-47.859,179.948,6.101,149.113
C04338=1158.222,13.354,-47.844,179.944,6.100,149.114
C04339=1158.228,13.105,-47.831,179.942,6.099,149.114
C04340=1158.233,12.855,-47.816,179.940,6.099,149.115
C04341=1158.238,12.605,-47.803,179.937,6.098,149.115
C04342=1158.244,12.356,-47.789,179.935,6.098,149.116
C04343=1158.248,12.107,-47.775,179.933,6.097,149.117
C04344=1158.253,11.857,-47.761,179.929,6.096,149.117
C04345=1158.258,11.608,-47.747,179.927,6.095,149.118
C04346=1158.264,11.358,-47.733,179.925,6.094,149.118
C04347=1158.269,11.108,-47.719,179.922,6.093,149.119
C04348=1158.274,10.859,-47.705,179.920,6.093,149.120
C04349=1158.278,10.609,-47.692,179.917,6.093,149.120
C04350=1158.284,10.359,-47.678,179.914,6.091,149.121
C04351=1158.289,10.110,-47.664,179.912,6.090,149.121
C04352=1158.294,9.860,-47.650,179.910,6.090,149.122
C04353=1158.299,9.610,-47.637,179.907,6.089,149.123
C04354=1158.304,9.361,-47.623,179.905,6.088,149.123
C04355=1158.309,9.112,-47.609,179.902,6.088,149.124
C04356=1158.315,8.862,-47.595,179.899,6.086,149.124
C04357=1158.319,8.613,-47.582,179.897,6.086,149.125
C04358=1158.324,8.363,-47.567,179.894,6.085,149.125
C04359=1158.330,8.113,-47.554,179.892,6.085,149.126
C04360=1158.335,7.864,-47.540,179.890,6.084,149.126
C04361=1158.340,7.615,-47.527,179.887,6.083,149.127
C04362=1158.345,7.365,-47.513,179.884,6.082,149.128
C04363=1158.350,7.115,-47.499,179.882,6.081,149.128
C04364=1158.356,6.866,-47.485,179.879,6.080,149.129
C04365=1158.360,6.616,-47.472,179.877,6.080,149.129
C04366=1158.366,6.367,-47.458,179.875,6.079,149.130
C04367=1158.371,6.116,-47.444,179.872,6.079,149.131
C04368=1158.376,5.868,-47.431,179.870,6.078,149.131
C04369=1158.381,5.617,-47.418,179.867,6.077,149.132
C04370=1158.386,5.368,-47.403,179.864,6.076,149.132
C04371=1158.391,5.119,-47.390,179.862,6.075,149.133
C04372=1158.396,4.869,-47.376,179.859,6.075,149.134
C04373=1158.402,4.620,-47.363,179.857,6.074,149.134
C04374=1158.406,4.370,-47.350,179.854,6.074,149.135
C04375=1158.412,4.121,-47.336,179.852,6.073,149.135
C04376=1158.416,3.871,-47.323,179.849,6.072,149.136
C04377=1158.422,3.622,-47.309,179.847,6.071,149.136
C04378=1158.427,3.371,-47.295,179.844,6.070,149.137
C04379=1158.431,3.122,-47.282,179.842,6.069,149.137
C04380=1158.437,2.872,-47.268,179.839,6.069,149.138
C04381=1158.442,2.622,-47.255,179.837,6.068,149.139
C04382=1158.447,2.373,-47.241,179.834,6.068,149.139
C04383=1158.453,2.104,-47.226,179.832,6.067,149.140
C04384=1158.458,1.834,-47.212,179.829,6.066,149.140
C04385=1158.464,1.565,-47.198,179.826,6.065,149.141
C04386=1158.469,1.296,-47.183,179.824,6.065,149.142
C04387=1158.475,1.046,-47.170,179.821,6.064,149.142
C04388=1158.479,0.796,-47.157,179.819,6.063,149.143
C04389=1158.485,0.547,-47.143,179.816,6.062,149.143
C04390=1158.489,0.297,-47.130,179.813,6.061,149.144
C04391=1158.495,0.048,-47.117,179.811,6.061,149.145
C04392=1158.500,-0.202,-47.103,179.808,6.060,149.145
C04393=1158.505,-0.451,-47.090,179.806,6.059,149.146
C04394=1158.510,-0.701,-47.076,179.804,6.059,149.146
C04395=1158.516,-0.950,-47.063,179.801,6.058,149.147
C04396=1158.521,-1.201,-47.050,179.799,6.058,149.148
C04397=1158.526,-1.449,-47.036,179.796,6.057,149.148
C04398=1158.531,-1.700,-47.023,179.794,6.056,149.149
C04399=1158.536,-1.949,-47.010,179.791,6.055,149.149
C04400=1158.542,-2.199,-46.997,179.789,6.054,149.150
C04401=1158.546,-2.448,-46.983,179.786,6.054,149.151
C04402=1158.552,-2.698,-46.970,179.784,6.053,149.151
C04403=1158.556,-2.948,-46.957,179.781,6.052,149.152
C04404=1158.561,-3.196,-46.944,179.779,6.052,149.152
C04405=1158.567,-3.447,-46.930,179.776,6.051,149.153
C04406=1158.572,-3.696,-46.918,179.774,6.050,149.153
C04407=1158.578,-3.946,-46.904,179.771,6.050,149.154
C04408=1158.582,-4.196,-46.891,179.769,6.049,149.155
C04409=1158.588,-4.445,-46.878,179.767,6.049,149.155
C04410=1158.592,-4.695,-46.865,179.764,6.048,149.156
C04411=1158.598,-4.944,-46.851,179.761,6.047,149.156
C04412=1158.603,-5.194,-46.839,179.759,6.046,149.157
C04413=1158.607,-5.443,-46.825,179.756,6.045,149.158
C04414=1158.613,-5.693,-46.812,179.754,6.045,149.158
C04415=1158.618,-5.943,-46.799,179.752,6.044,149.159
C04416=1158.624,-6.192,-46.786,179.749,6.044,149.159
C04417=1158.629,-6.442,-46.773,179.747,6.043,149.160
C04418=1158.633,-6.692,-46.760,179.744,6.042,149.161
C04419=1158.639,-6.941,-46.747,179.742,6.042,149.161
C04420=1158.644,-7.190,-46.734,179.739,6.041,149.162
C04421=1158.648,-7.440,-46.721,179.737,6.040,149.162
C04422=1158.654,-7.690,-46.708,179.734,6.040,149.163
C04423=1158.659,-7.940,-46.695,179.732,6.039,149.163
C04424=1158.664,-8.189,-46.682,179.730,6.039,149.164
C04425=1158.670,-8.439,-46.669,179.727,6.038,149.165
C04426=1158.674,-8.689,-46.656,179.724,6.037,149.165
C04427=1158.679,-8.938,-46.643,179.721,6.036,149.166
C04428=1158.685,-9.188,-46.630,179.719,6.035,149.166
C04429=1158.690,-9.438,-46.617,179.717,6.035,149.167
C04430=1158.695,-9.687,-46.604,179.714,6.034,149.167
C04431=1158.701,-9.937,-46.591,179.712,6.034,149.168
C04432=1158.705,-10.187,-46.578,179.710,6.033,149.169
C04433=1158.710,-10.435,-46.565,179.707,6.032,149.169
C04434=1158.716,-10.685,-46.552,179.705,6.032,149.170
C04435=1158.721,-10.934,-46.539,179.702,6.031,149.170
C04436=1158.726,-11.184,-46.526,179.700,6.030,149.171
C04437=1158.731,-11.434,-46.514,179.697,6.030,149.172
C04438=1158.737,-11.683,-46.500,179.695,6.029,149.172
C04439=1158.741,-11.934,-46.488,179.692,6.029,149.173
C04440=1158.747,-12.183,-46.476,179.690,6.028,149.173
C04441=1158.752,-12.432,-46.463,179.688,6.027,149.174
C04442=1158.757,-12.683,-46.449,179.685,6.027,149.175
C04443=1158.762,-12.932,-46.437,179.683,6.026,149.175
C04444=1158.767,-13.181,-46.424,179.680,6.026,149.176
C04445=1158.772,-13.431,-46.412,179.678,6.025,149.176
C04446=1158.777,-13.681,-46.399,179.675,6.024,149.177
C04447=1158.783,-13.930,-46.385,179.673,6.024,149.177
C04448=1158.788,-14.180,-46.373,179.670,6.023,149.178
C04449=1158.793,-14.429,-46.360,179.668,6.022,149.179
C04450=1158.797,-14.679,-46.347,179.666,6.022,149.179
C04451=1158.803,-14.929,-46.335,179.663,6.021,149.180
C04452=1158.809,-15.179,-46.322,179.661,6.021,149.180
C04453=1158.814,-15.428,-46.310,179.659,6.020,149.181
C04454=1158.818,-15.678,-46.297,179.656,6.019,149.182
C04455=1158.824,-15.927,-46.284,179.654,6.019,149.182
C04456=1158.829,-16.177,-46.271,179.651,6.018,149.183
C04457=1158.834,-16.426,-46.259,179.648,6.018,149.183
C04458=1158.840,-16.676,-46.246,179.646,6.017,149.184
C04459=1158.844,-16.926,-46.233,179.644,6.017,149.185
C04460=1158.850,-17.175,-46.221,179.641,6.016,149.185
C04461=1158.855,-17.425,-46.208,179.639,6.015,149.186
C04462=1158.860,-17.674,-46.196,179.637,6.014,149.186
C04463=1158.865,-17.924,-46.184,179.634,6.014,149.187
C04464=1158.870,-18.174,-46.171,179.632,6.013,149.187
C04465=1158.876,-18.424,-46.157,179.629,6.013,149.188
C04466=1158.881,-18.673,-46.145,179.627,6.012,149.189
C04467=1158.886,-18.923,-46.133,179.624,6.012,149.189
C04468=1158.891,-19.172,-46.120,179.622,6.011,149.190
C04469=1158.896,-19.422,-46.108,179.619,6.010,149.190
C04470=1158.901,-19.672,-46.095,179.617,6.009,149.191
C04471=1158.906,-19.922,-46.083,179.615,6.009,149.192
C04472=1158.912,-20.171,-46.070,179.612,6.008,149.192
C04473=1158.917,-20.420,-46.058,179.610,6.008,149.193
C04474=1158.922,-20.670,-46.046,179.607,6.007,149.193
C04475=1158.927,-20.919,-46.033,179.605,6.007,149.194
C04476=1158.932,-21.169,-46.020,179.602,6.006,149.195
C04477=1158.937,-21.419,-46.008,179.600,6.005,149.195
C04478=1158.942,-21.669,-45.996,179.597,6.005,149.196
C04479=1158.948,-21.918,-45.983,179.595,6.004,149.196
C04480=1158.954,-22.168,-45.971,179.593,6.004,149.197
C04481=1158.959,-22.418,-45.958,179.590,6.003,149.197
C04482=1158.964,-22.667,-45.946,179.588,6.002,149.198
C04483=1158.969,-22.917,-45.934,179.586,6.002,149.199
C04484=1158.974,-23.166,-45.921,179.583,6.001,149.199
C04485=1158.979,-23.417,-45.909,179.581,6.000,149.200
C04486=1158.984,-23.666,-45.896,179.578,6.000,149.200
C04487=1158.990,-23.936,-45.884,179.575,6.000,149.201
C04488=1158.995,-24.206,-45.870,179.573,5.999,149.202
C04489=1159.001,-24.476,-45.857,179.571,5.998,149.202
C04490=1159.007,-24.745,-45.843,179.567,5.997,149.203
C04491=1159.012,-24.995,-45.831,179.566,5.997,149.204
C04492=1159.017,-25.244,-45.819,179.563,5.997,149.204
C04493=1159.022,-25.495,-45.806,179.561,5.996,149.205
C04494=1159.027,-25.744,-45.794,179.558,5.995,149.205
C04495=1159.032,-25.994,-45.782,179.556,5.995,149.206
C04496=1159.037,-26.243,-45.770,179.553,5.994,149.207
C04497=1159.043,-26.493,-45.758,179.551,5.994,149.207
C04498=1159.048,-26.743,-45.745,179.548,5.993,149.208
C04499=1159.053,-26.993,-45.733,179.546,5.993,149.208
C04500=1159.058,-27.242,-45.721,179.544,5.992,149.209
C04501=1159.064,-27.492,-45.709,179.541,5.991,149.210
C04502=1159.069,-27.741,-45.696,179.539,5.990,149.210
C04503=1159.074,-27.991,-45.684,179.536,5.990,149.211
C04504=1159.079,-28.240,-45.672,179.534,5.989,149.211
C04505=1159.084,-28.490,-45.661,179.531,5.989,149.212
C04506=1159.090,-28.740,-45.649,179.529,5.988,149.212
C04507=1159.095,-28.989,-45.636,179.526,5.988,149.213
C04508=1159.100,-29.239,-45.624,179.524,5.987,149.214
C04509=1159.105,-29.489,-45.612,179.522,5.986,149.214
C04510=1159.111,-29.738,-45.600,179.520,5.986,149.215
C04511=1159.116,-29.988,-45.587,179.517,5.986,149.215
C04512=1159.120,-30.237,-45.576,179.515,5.985,149.216
C04513=1159.126,-30.487,-45.564,179.513,5.985,149.217
C04514=1159.131,-30.737,-45.551,179.510,5.984,149.217
C04515=1159.136,-30.987,-45.539,179.508,5.983,149.218
C04516=1159.142,-31.237,-45.528,179.505,5.983,149.218
C04517=1159.146,-31.486,-45.516,179.503,5.982,149.219
C04518=1159.152,-31.735,-45.504,179.500,5.982,149.220
C04519=1159.157,-31.985,-45.492,179.498,5.981,149.220
C04520=1159.162,-32.235,-45.479,179.495,5.981,149.221
C04521=1159.168,-32.485,-45.467,179.493,5.980,149.221
C04522=1159.172,-32.734,-45.456,179.490,5.979,149.222
C04523=1159.178,-32.984,-45.443,179.488,5.979,149.222
C04524=1159.183,-33.234,-45.432,179.486,5.979,149.223
C04525=1159.188,-33.483,-45.420,179.484,5.978,149.224
C04526=1159.194,-33.733,-45.408,179.481,5.978,149.224
C04527=1159.198,-33.982,-45.396,179.479,5.977,149.225
C04528=1159.204,-34.232,-45.384,179.477,5.977,149.225
C04529=1159.209,-34.482,-45.372,179.474,5.976,149.226
C04530=1159.214,-34.732,-45.360,179.472,5.975,149.227
C04531=1159.219,-34.981,-45.348,179.469,5.974,149.227
C04532=1159.224,-35.231,-45.336,179.467,5.974,149.228
C04533=1159.230,-35.481,-45.324,179.465,5.973,149.228
C04534=1159.234,-35.731,-45.313,179.463,5.974,149.229
C04535=1159.240,-35.979,-45.301,179.460,5.973,149.229
C04536=1159.246,-36.229,-45.289,179.458,5.972,149.230
C04537=1159.251,-36.479,-45.277,179.456,5.972,149.231
C04538=1159.256,-36.729,-45.266,179.453,5.971,149.231
C04539=1159.261,-36.979,-45.254,179.451,5.970,149.232
C04540=1159.267,-37.229,-45.242,179.448,5.970,149.233
C04541=1159.271,-37.478,-45.230,179.446,5.969,149.233
C04542=1159.276,-37.728,-45.218,179.443,5.969,149.234
C04543=1159.282,-37.978,-45.206,179.441,5.968,149.234
C04544=1159.287,-38.227,-45.195,179.439,5.968,149.235
C04545=1159.293,-38.476,-45.183,179.437,5.968,149.235
C04546=1159.298,-38.726,-45.171,179.434,5.967,149.236
C04547=1159.303,-38.976,-45.160,179.432,5.966,149.237
C04548=1159.308,-39.226,-45.148,179.429,5.966,149.237
C04549=1159.313,-39.475,-45.136,179.427,5.966,149.238
C04550=1159.318,-39.725,-45.124,179.424,5.965,149.238
C04551=1159.323,-39.975,-45.113,179.422,5.964,149.239
C04552=1159.329,-40.224,-45.102,179.420,5.964,149.240
C04553=1159.334,-40.474,-45.090,179.417,5.964,149.240
C04554=1159.339,-40.724,-45.078,179.415,5.963,149.241
C04555=1159.344,-40.973,-45.067,179.413,5.963,149.241
C04556=1159.350,-41.223,-45.055,179.410,5.962,149.242
C04557=1159.355,-41.473,-45.043,179.408,5.961,149.243
C04558=1159.360,-41.722,-45.032,179.406,5.961,149.243
C04559=1159.366,-41.972,-45.020,179.403,5.960,149.244
C04560=1159.370,-42.222,-45.009,179.401,5.960,149.244
C04561=1159.376,-42.472,-44.997,179.399,5.960,149.245
C04562=1159.381,-42.721,-44.986,179.396,5.959,149.245
C04563=1159.386,-42.971,-44.974,179.394,5.959,149.246
C04564=1159.391,-43.220,-44.963,179.392,5.958,149.247
C04565=1159.397,-43.470,-44.951,179.389,5.957,149.247
C04566=1159.402,-43.720,-44.939,179.387,5.957,149.248
C04567=1159.407,-43.970,-44.928,179.384,5.956,149.249
C04568=1159.412,-44.219,-44.916,179.383,5.956,149.249
C04569=1159.418,-44.468,-44.905,179.380,5.956,149.250
C04570=1159.423,-44.718,-44.893,179.378,5.955,149.250
C04571=1159.428,-44.968,-44.882,179.375,5.955,149.251
C04572=1159.433,-45.218,-44.870,179.373,5.954,149.251
C04573=1159.438,-45.468,-44.859,179.370,5.953,149.252
C04574=1159.444,-45.717,-44.848,179.369,5.953,149.253
C04575=1159.449,-45.967,-44.836,179.366,5.953,149.253
C04576=1159.454,-46.217,-44.824,179.364,5.952,149.254
C04577=1159.459,-46.467,-44.813,179.361,5.952,149.254
C04578=1159.465,-46.716,-44.802,179.359,5.951,149.255
C04579=1159.470,-46.965,-44.790,179.356,5.951,149.256
C04580=1159.475,-47.215,-44.779,179.354,5.950,149.256
C04581=1159.480,-47.466,-44.768,179.352,5.950,149.257
C04582=1159.485,-47.715,-44.757,179.350,5.949,149.257
C04583=1159.491,-47.964,-44.745,179.347,5.949,149.258
C04584=1159.495,-48.214,-44.734,179.345,5.948,149.258
C04585=1159.501,-48.464,-44.722,179.342,5.948,149.259
C04586=1159.506,-48.713,-44.711,179.340,5.947,149.260
C04587=1159.512,-48.964,-44.700,179.338,5.947,149.260
C04588=1159.517,-49.213,-44.689,179.336,5.947,149.261
C04589=1159.522,-49.463,-44.677,179.333,5.946,149.261
C04590=1159.527,-49.712,-44.666,179.331,5.945,149.262
C04591=1159.533,-49.983,-44.654,179.328,5.945,149.263
C04592=1159.539,-50.253,-44.642,179.326,5.945,149.263
C04593=1159.545,-50.524,-44.629,179.323,5.944,149.264
C04594=1159.549,-50.794,-44.617,179.321,5.943,149.265
C04595=1159.556,-51.044,-44.606,179.319,5.943,149.265
C04596=1159.560,-51.294,-44.595,179.317,5.943,149.266
C04597=1159.566,-51.544,-44.583,179.314,5.942,149.266
C04598=1159.571,-51.793,-44.572,179.312,5.942,149.267
C04599=1159.576,-52.043,-44.562,179.309,5.941,149.267
C04600=1159.582,-52.293,-44.550,179.307,5.941,149.268
C04601=1159.586,-52.542,-44.538,179.305,5.940,149.269
C04602=1159.592,-52.792,-44.528,179.303,5.940,149.269
C04603=1159.597,-53.042,-44.516,179.300,5.939,149.270
C04604=1159.602,-53.292,-44.505,179.298,5.939,149.270
C04605=1159.608,-53.541,-44.495,179.295,5.938,149.271
C04606=1159.613,-53.791,-44.483,179.293,5.938,149.272
C04607=1159.618,-54.041,-44.472,179.291,5.938,149.272
C04608=1159.623,-54.290,-44.461,179.289,5.937,149.273
C04609=1159.629,-54.540,-44.449,179.286,5.937,149.273
C04610=1159.633,-54.790,-44.438,179.284,5.936,149.274
C04611=1159.639,-55.039,-44.428,179.282,5.935,149.274
C04612=1159.644,-55.289,-44.417,179.279,5.936,149.275
C04613=1159.650,-55.539,-44.406,179.277,5.935,149.276
C04614=1159.655,-55.788,-44.395,179.275,5.935,149.276
C04615=1159.659,-56.038,-44.383,179.272,5.934,149.277
C04616=1159.665,-56.288,-44.373,179.270,5.933,149.278
C04617=1159.670,-56.537,-44.361,179.268,5.933,149.278
C04618=1159.675,-56.788,-44.351,179.265,5.933,149.279
C04619=1159.681,-57.037,-44.340,179.263,5.932,149.279
C04620=1159.685,-57.286,-44.328,179.261,5.932,149.280
C04621=1159.692,-57.536,-44.318,179.258,5.931,149.280
C04622=1159.696,-57.786,-44.306,179.256,5.931,149.281
C04623=1159.701,-58.036,-44.296,179.254,5.931,149.282
C04624=1159.707,-58.285,-44.285,179.252,5.930,149.282
C04625=1159.712,-58.535,-44.274,179.249,5.929,149.283
C04626=1159.718,-58.784,-44.263,179.247,5.929,149.283
C04627=1159.723,-59.035,-44.252,179.245,5.929,149.284
C04628=1159.727,-59.284,-44.241,179.243,5.928,149.284
C04629=1159.733,-59.534,-44.231,179.240,5.928,149.285
C04630=1159.739,-59.784,-44.219,179.238,5.927,149.286
C04631=1159.744,-60.033,-44.209,179.236,5.927,149.286
C04632=1159.749,-60.283,-44.197,179.234,5.927,149.287
C04633=1159.754,-60.533,-44.187,179.231,5.926,149.287
C04634=1159.759,-60.782,-44.176,179.229,5.925,149.288
C04635=1159.764,-61.032,-44.165,179.226,5.925,149.289
C04636=1159.770,-61.282,-44.154,179.225,5.925,149.289
C04637=1159.775,-61.532,-44.143,179.222,5.925,149.290
C04638=1159.781,-61.781,-44.133,179.220,5.924,149.290
C04639=1159.785,-62.031,-44.122,179.217,5.923,149.291
C04640=1159.791,-62.281,-44.111,179.216,5.923,149.292
C04641=1159.796,-62.530,-44.100,179.213,5.923,149.292
C04642=1159.801,-62.780,-44.090,179.211,5.922,149.293
C04643=1159.807,-63.030,-44.079,179.208,5.921,149.293
C04644=1159.812,-63.280,-44.067,179.206,5.922,149.294
C04645=1159.817,-63.529,-44.057,179.204,5.921,149.294
C04646=1159.822,-63.780,-44.047,179.202,5.921,149.295
C04647=1159.828,-64.029,-44.036,179.199,5.920,149.296
C04648=1159.833,-64.279,-44.025,179.197,5.920,149.296
C04649=1159.838,-64.528,-44.014,179.195,5.920,149.297
C04650=1159.843,-64.778,-44.004,179.192,5.919,149.297
C04651=1159.848,-65.028,-43.993,179.190,5.918,149.298
C04652=1159.853,-65.277,-43.982,179.188,5.919,149.299
C04653=1159.860,-65.527,-43.971,179.186,5.918,149.299
C04654=1159.865,-65.777,-43.961,179.183,5.918,149.300
C04655=1159.870,-66.027,-43.951,179.181,5.917,149.300
C04656=1159.875,-66.276,-43.939,179.180,5.917,149.301
C04657=1159.880,-66.526,-43.929,179.177,5.916,149.301
C04658=1159.886,-66.776,-43.919,179.175,5.916,149.302
C04659=1159.891,-67.025,-43.908,179.172,5.915,149.303
C04660=1159.896,-67.275,-43.897,179.170,5.915,149.303
C04661=1159.901,-67.525,-43.887,179.168,5.915,149.304
C04662=1159.907,-67.774,-43.877,179.166,5.914,149.304
C04663=1159.912,-68.024,-43.865,179.163,5.914,149.305
C04664=1159.917,-68.274,-43.855,179.161,5.914,149.306
C04665=1159.922,-68.524,-43.845,179.159,5.913,149.306
C04666=1159.928,-68.773,-43.834,179.156,5.912,149.307
C04667=1159.932,-69.023,-43.823,179.154,5.912,149.307
C04668=1159.938,-69.273,-43.813,179.152,5.912,149.308
C04669=1159.944,-69.522,-43.803,179.150,5.911,149.308
C04670=1159.949,-69.772,-43.792,179.147,5.911,149.309
C04671=1159.954,-70.022,-43.782,179.145,5.910,149.310
C04672=1159.959,-70.272,-43.771,179.143,5.911,149.310
C04673=1159.965,-70.521,-43.760,179.141,5.910,149.311
C04674=1159.970,-70.771,-43.750,179.138,5.909,149.311
C04675=1159.975,-71.021,-43.740,179.137,5.909,149.312
C04676=1159.981,-71.270,-43.729,179.134,5.909,149.312
C04677=1159.986,-71.521,-43.719,179.132,5.908,149.313
C04678=1159.991,-71.770,-43.709,179.130,5.907,149.314
C04679=1159.996,-72.020,-43.697,179.127,5.908,149.314
C04680=1160.002,-72.269,-43.687,179.125,5.907,149.315
C04681=1160.007,-72.519,-43.677,179.123,5.907,149.316
C04682=1160.012,-72.769,-43.666,179.121,5.907,149.316
C04683=1160.018,-73.019,-43.656,179.119,5.906,149.316
C04684=1160.022,-73.269,-43.646,179.116,5.905,149.317
C04685=1160.028,-73.518,-43.636,179.114,5.905,149.318
C04686=1160.033,-73.768,-43.626,179.112,5.905,149.318
C04687=1160.038,-74.018,-43.615,179.110,5.904,149.319
C04688=1160.044,-74.268,-43.605,179.107,5.904,149.320
C04689=1160.049,-74.517,-43.595,179.105,5.904,149.320
C04690=1160.054,-74.767,-43.584,179.103,5.904,149.321
C04691=1160.060,-75.017,-43.574,179.101,5.903,149.321
C04692=1160.065,-75.266,-43.563,179.098,5.902,149.322
C04693=1160.070,-75.516,-43.552,179.096,5.902,149.322
C04694=1160.075,-75.765,-43.543,179.094,5.902,149.323
C04695=1160.081,-76.037,-43.531,179.091,5.901,149.324
C04696=1160.088,-76.308,-43.520,179.089,5.901,149.324
C04697=1160.093,-76.579,-43.509,179.087,5.900,149.325
C04698=1160.099,-76.851,-43.498,179.084,5.900,149.326
C04699=1160.104,-77.100,-43.488,179.082,5.900,149.326
C04700=1160.109,-77.349,-43.478,179.080,5.899,149.327
C04701=1160.114,-77.600,-43.467,179.078,5.899,149.327
C04702=1160.120,-77.850,-43.458,179.076,5.899,149.328
C04703=1160.126,-78.099,-43.448,179.073,5.898,149.328
C04704=1160.131,-78.350,-43.437,179.071,5.897,149.329
C04705=1160.136,-78.599,-43.427,179.069,5.898,149.330
C04706=1160.141,-78.848,-43.417,179.067,5.897,149.330
C04707=1160.146,-79.099,-43.407,179.064,5.897,149.331
C04708=1160.152,-79.348,-43.396,179.062,5.897,149.331
C04709=1160.157,-79.598,-43.386,179.060,5.896,149.332
C04710=1160.162,-79.847,-43.377,179.058,5.895,149.332
C04711=1160.167,-80.097,-43.366,179.056,5.895,149.333
C04712=1160.173,-80.347,-43.356,179.053,5.895,149.334
C04713=1160.178,-80.596,-43.346,179.051,5.894,149.334
C04714=1160.183,-80.847,-43.336,179.050,5.894,149.335
C04715=1160.189,-81.096,-43.326,179.047,5.894,149.335
C04716=1160.194,-81.346,-43.316,179.045,5.893,149.336
C04717=1160.200,-81.596,-43.306,179.043,5.894,149.336
C04718=1160.204,-81.845,-43.296,179.040,5.893,149.337
C04719=1160.210,-82.095,-43.285,179.038,5.892,149.338
C04720=1160.215,-82.345,-43.275,179.036,5.892,149.338
C04721=1160.221,-82.595,-43.266,179.034,5.892,149.339
C04722=1160.225,-82.845,-43.256,179.031,5.891,149.339
C04723=1160.231,-83.094,-43.246,179.030,5.891,149.340
C04724=1160.237,-83.344,-43.235,179.027,5.891,149.341
C04725=1160.242,-83.593,-43.225,179.025,5.890,149.341
C04726=1160.246,-83.843,-43.215,179.023,5.890,149.341
C04727=1160.252,-84.093,-43.206,179.021,5.890,149.342
C04728=1160.258,-84.343,-43.195,179.018,5.889,149.343
C04729=1160.263,-84.592,-43.186,179.016,5.889,149.343
C04730=1160.268,-84.842,-43.175,179.014,5.889,149.344
C04731=1160.274,-85.093,-43.166,179.012,5.888,149.344
C04732=1160.279,-85.342,-43.156,179.010,5.888,149.345
C04733=1160.284,-85.591,-43.146,179.008,5.887,149.346
C04734=1160.289,-85.842,-43.135,179.005,5.887,149.346
C04735=1160.294,-86.091,-43.126,179.003,5.887,149.347
C04736=1160.300,-86.341,-43.116,179.001,5.886,149.347
C04737=1160.306,-86.590,-43.106,178.998,5.886,149.348
C04738=1160.310,-86.840,-43.096,178.997,5.886,149.348
C04739=1160.316,-87.091,-43.087,178.995,5.885,149.349
C04740=1160.321,-87.340,-43.077,178.992,5.885,149.350
C04741=1160.326,-87.589,-43.067,178.990,5.885,149.350
C04742=1160.332,-87.840,-43.057,178.988,5.884,149.351
C04743=1160.337,-88.089,-43.048,178.986,5.884,149.351
C04744=1160.342,-88.339,-43.037,178.984,5.884,149.352
C04745=1160.347,-88.589,-43.028,178.981,5.883,149.352
C04746=1160.353,-88.838,-43.018,178.979,5.883,149.353
C04747=1160.358,-89.088,-43.008,178.977,5.883,149.354
C04748=1160.363,-89.338,-42.999,178.975,5.882,149.354
C04749=1160.369,-89.587,-42.989,178.973,5.882,149.355
C04750=1160.373,-89.837,-42.979,178.971,5.882,149.355
C04751=1160.379,-90.087,-42.969,178.968,5.881,149.356
C04752=1160.385,-90.337,-42.959,178.967,5.881,149.356
C04753=1160.390,-90.587,-42.950,178.964,5.881,149.357
C04754=1160.396,-90.836,-42.940,178.962,5.880,149.358
C04755=1160.400,-91.086,-42.930,178.960,5.880,149.358
C04756=1160.406,-91.336,-42.921,178.958,5.880,149.359
C04757=1160.411,-91.586,-42.911,178.955,5.879,149.359
C04758=1160.417,-91.836,-42.901,178.953,5.879,149.360
C04759=1160.421,-92.085,-42.892,178.951,5.878,149.360
C04760=1160.427,-92.335,-42.881,178.950,5.878,149.361
C04761=1160.433,-92.585,-42.872,178.947,5.878,149.362
C04762=1160.438,-92.834,-42.862,178.945,5.877,149.362
C04763=1160.444,-93.084,-42.853,178.943,5.878,149.363
C04764=1160.449,-93.333,-42.843,178.940,5.877,149.363
C04765=1160.454,-93.584,-42.833,178.938,5.876,149.364
C04766=1160.459,-93.834,-42.824,178.936,5.877,149.364
C04767=1160.465,-94.084,-42.814,178.934,5.876,149.365
C04768=1160.469,-94.333,-42.805,178.932,5.876,149.365
C04769=1160.475,-94.583,-42.795,178.930,5.875,149.366
C04770=1160.480,-94.832,-42.786,178.928,5.875,149.367
C04771=1160.486,-95.082,-42.776,178.926,5.875,149.367
C04772=1160.491,-95.332,-42.766,178.923,5.874,149.368
C04773=1160.497,-95.582,-42.757,178.921,5.874,149.368
C04774=1160.502,-95.831,-42.747,178.919,5.874,149.369
C04775=1160.507,-96.081,-42.738,178.917,5.873,149.370
C04776=1160.512,-96.331,-42.728,178.915,5.873,149.370
C04777=1160.517,-96.581,-42.719,178.913,5.873,149.371
C04778=1160.523,-96.831,-42.709,178.910,5.872,149.371
C04779=1160.528,-97.080,-42.700,178.909,5.872,149.372
C04780=1160.534,-97.331,-42.690,178.906,5.872,149.372
C04781=1160.539,-97.580,-42.681,178.904,5.872,149.373
C04782=1160.545,-97.830,-42.671,178.902,5.871,149.373
C04783=1160.549,-98.079,-42.662,178.900,5.871,149.374
C04784=1160.555,-98.329,-42.653,178.898,5.871,149.375
C04785=1160.560,-98.579,-42.643,178.896,5.870,149.375
C04786=1160.565,-98.828,-42.634,178.894,5.870,149.376
C04787=1160.571,-99.079,-42.624,178.892,5.870,149.376
C04788=1160.576,-99.328,-42.615,178.889,5.869,149.377
C04789=1160.582,-99.578,-42.605,178.887,5.869,149.377
C04790=1160.587,-99.828,-42.596,178.885,5.868,149.378
C04791=1160.592,-100.077,-42.587,178.883,5.868,149.378
C04792=1160.598,-100.327,-42.577,178.881,5.868,149.379
C04793=1160.603,-100.577,-42.568,178.879,5.867,149.380
C04794=1160.608,-100.826,-42.559,178.877,5.867,149.380
C04795=1160.614,-101.077,-42.549,178.874,5.867,149.381
C04796=1160.619,-101.326,-42.540,178.873,5.867,149.381
C04797=1160.625,-101.576,-42.530,178.871,5.866,149.382
C04798=1160.630,-101.826,-42.521,178.868,5.866,149.382
C04799=1160.635,-102.098,-42.511,178.866,5.866,149.383
C04800=1160.641,-102.370,-42.501,178.864,5.866,149.384
C04801=1160.646,-102.642,-42.490,178.861,5.865,149.384
C04802=1160.653,-102.914,-42.481,178.859,5.865,149.385
C04803=1160.658,-103.163,-42.471,178.857,5.864,149.385
C04804=1160.663,-103.413,-42.462,178.854,5.864,149.386
C04805=1160.669,-103.663,-42.453,178.853,5.864,149.387
C04806=1160.674,-103.913,-42.444,178.851,5.863,149.387
C04807=1160.679,-104.162,-42.434,178.849,5.863,149.388
C04808=1160.685,-104.412,-42.425,178.846,5.863,149.388
C04809=1160.690,-104.662,-42.416,178.844,5.862,149.389
C04810=1160.696,-104.912,-42.407,178.843,5.862,149.389
C04811=1160.700,-105.161,-42.397,178.840,5.862,149.390
C04812=1160.706,-105.411,-42.388,178.838,5.862,149.390
C04813=1160.712,-105.661,-42.379,178.836,5.861,149.391
C04814=1160.717,-105.911,-42.370,178.834,5.862,149.392
C04815=1160.722,-106.161,-42.361,178.832,5.861,149.392
C04816=1160.727,-106.410,-42.351,178.830,5.860,149.393
C04817=1160.733,-106.660,-42.342,178.828,5.860,149.393
C04818=1160.738,-106.910,-42.333,178.825,5.860,149.394
C04819=1160.743,-107.160,-42.324,178.824,5.860,149.394
C04820=1160.749,-107.410,-42.315,178.821,5.859,149.395
C04821=1160.754,-107.659,-42.305,178.820,5.859,149.395
C04822=1160.759,-107.909,-42.296,178.817,5.859,149.396
C04823=1160.764,-108.159,-42.287,178.816,5.859,149.396
C04824=1160.771,-108.408,-42.278,178.813,5.858,149.397
C04825=1160.776,-108.658,-42.269,178.811,5.857,149.398
C04826=1160.781,-108.908,-42.260,178.809,5.857,149.398
C04827=1160.786,-109.158,-42.251,178.807,5.857,149.399
C04828=1160.791,-109.408,-42.242,178.805,5.857,149.399
C04829=1160.797,-109.657,-42.232,178.803,5.856,149.400
C04830=1160.802,-109.907,-42.223,178.801,5.856,149.400
C04831=1160.807,-110.157,-42.214,178.799,5.856,149.401
C04832=1160.812,-110.407,-42.206,178.796,5.855,149.402
C04833=1160.817,-110.657,-42.197,178.795,5.855,149.402
C04834=1160.824,-110.906,-42.188,178.792,5.855,149.403
C04835=1160.829,-111.156,-42.179,178.790,5.855,149.403
C04836=1160.834,-111.406,-42.170,178.788,5.854,149.404
C04837=1160.839,-111.656,-42.161,178.786,5.855,149.404
C04838=1160.845,-111.906,-42.152,178.784,5.854,149.405
C04839=1160.850,-112.156,-42.143,178.782,5.854,149.405
C04840=1160.856,-112.406,-42.134,178.780,5.853,149.406
C04841=1160.861,-112.656,-42.125,178.778,5.854,149.407
C04842=1160.867,-112.905,-42.116,178.776,5.853,149.407
C04843=1160.872,-113.155,-42.107,178.774,5.852,149.408
C04844=1160.877,-113.404,-42.098,178.772,5.852,149.408
C04845=1160.882,-113.654,-42.089,178.769,5.852,149.409
C04846=1160.887,-113.904,-42.081,178.768,5.852,149.409
C04847=1160.893,-114.154,-42.071,178.766,5.851,149.410
C04848=1160.899,-114.403,-42.063,178.764,5.851,149.410
C04849=1160.904,-114.653,-42.054,178.761,5.851,149.411
C04850=1160.909,-114.903,-42.045,178.760,5.851,149.411
C04851=1160.914,-115.153,-42.036,178.758,5.850,149.412
C04852=1160.920,-115.403,-42.027,178.755,5.850,149.413
C04853=1160.925,-115.653,-42.018,178.753,5.850,149.413
C04854=1160.931,-115.902,-42.010,178.752,5.850,149.414
C04855=1160.936,-116.152,-42.001,178.750,5.849,149.414
C04856=1160.941,-116.402,-41.992,178.747,5.848,149.415
C04857=1160.947,-116.652,-41.982,178.745,5.849,149.415
C04858=1160.952,-116.902,-41.973,178.743,5.848,149.416
C04859=1160.958,-117.151,-41.965,178.741,5.848,149.416
C04860=1160.963,-117.401,-41.956,178.739,5.847,149.417
C04861=1160.968,-117.650,-41.947,178.737,5.847,149.417
C04862=1160.974,-117.901,-41.939,178.735,5.847,149.418
C04863=1160.979,-118.151,-41.930,178.733,5.847,149.418
C04864=1160.984,-118.400,-41.921,178.731,5.846,149.419
C04865=1160.990,-118.650,-41.912,178.729,5.846,149.420
C04866=1160.995,-118.900,-41.904,178.727,5.846,149.420
C04867=1161.000,-119.149,-41.895,178.725,5.846,149.421
C04868=1161.005,-119.399,-41.886,178.723,5.845,149.421
C04869=1161.011,-119.648,-41.877,178.721,5.845,149.422
C04870=1161.016,-119.899,-41.869,178.719,5.845,149.422
C04871=1161.022,-120.149,-41.860,178.717,5.845,149.423
C04872=1161.027,-120.399,-41.851,178.715,5.844,149.423
C04873=1161.032,-120.648,-41.843,178.713,5.844,149.424
C04874=1161.038,-120.898,-41.834,178.711,5.844,149.424
C04875=1161.043,-121.147,-41.825,178.709,5.844,149.425
C04876=1161.048,-121.398,-41.817,178.706,5.843,149.426
C04877=1161.054,-121.647,-41.808,178.705,5.843,149.426
C04878=1161.059,-121.897,-41.799,178.703,5.842,149.427
C04879=1161.064,-122.147,-41.790,178.700,5.842,149.427
C04880=1161.070,-122.397,-41.782,178.698,5.842,149.428
C04881=1161.076,-122.646,-41.774,178.696,5.841,149.428
C04882=1161.081,-122.896,-41.765,178.695,5.841,149.429
C04883=1161.086,-123.146,-41.756,178.692,5.841,149.429
C04884=1161.091,-123.396,-41.747,178.691,5.841,149.430
C04885=1161.097,-123.646,-41.739,178.688,5.840,149.430
C04886=1161.102,-123.896,-41.730,178.687,5.840,149.431
C04887=1161.108,-124.145,-41.721,178.684,5.840,149.431
C04888=1161.113,-124.394,-41.713,178.683,5.840,149.432
C04889=1161.118,-124.645,-41.705,178.680,5.839,149.433
C04890=1161.123,-124.895,-41.696,178.678,5.839,149.433
C04891=1161.128,-125.144,-41.688,178.676,5.839,149.434
C04892=1161.134,-125.394,-41.680,178.675,5.839,149.434
C04893=1161.140,-125.644,-41.671,178.672,5.838,149.435
C04894=1161.145,-125.894,-41.662,178.670,5.838,149.435
C04895=1161.151,-126.144,-41.654,178.668,5.838,149.436
C04896=1161.156,-126.394,-41.645,178.667,5.838,149.436
C04897=1161.161,-126.643,-41.636,178.664,5.837,149.437
C04898=1161.167,-126.893,-41.628,178.663,5.837,149.437
C04899=1161.172,-127.143,-41.620,178.660,5.837,149.438
C04900=1161.177,-127.393,-41.611,178.659,5.837,149.438
C04901=1161.183,-127.642,-41.603,178.656,5.836,149.439
C04902=1161.188,-127.892,-41.595,178.655,5.836,149.439
C04903=1160.767,-127.903,-41.636,178.651,5.839,149.441
C04904=1160.762,-127.654,-41.645,178.653,5.840,149.441
C04905=1160.756,-127.404,-41.652,178.655,5.840,149.440
C04906=1160.751,-127.154,-41.661,178.657,5.840,149.440
C04907=1160.746,-126.904,-41.670,178.659,5.840,149.439
C04908=1160.740,-126.654,-41.678,178.661,5.841,149.439
C04909=1160.734,-126.404,-41.687,178.663,5.841,149.438
C04910=1160.729,-126.155,-41.696,178.665,5.842,149.438
C04911=1160.723,-125.905,-41.704,178.667,5.841,149.437
C04912=1160.718,-125.655,-41.713,178.669,5.842,149.436
C04913=1160.714,-125.405,-41.721,178.671,5.842,149.436
C04914=1160.708,-125.156,-41.730,178.673,5.843,149.435
C04915=1160.702,-124.906,-41.738,178.675,5.843,149.435
C04916=1160.697,-124.656,-41.746,178.677,5.843,149.434
C04917=1160.692,-124.406,-41.755,178.679,5.843,149.434
C04918=1160.686,-124.156,-41.763,178.681,5.844,149.433
C04919=1160.681,-123.906,-41.772,178.683,5.844,149.433
C04920=1160.676,-123.657,-41.781,178.685,5.844,149.432
C04921=1160.670,-123.407,-41.790,178.687,5.844,149.432
C04922=1160.664,-123.157,-41.798,178.689,5.845,149.431
C04923=1160.659,-122.907,-41.807,178.691,5.845,149.431
C04924=1160.654,-122.657,-41.815,178.693,5.845,149.430
C04925=1160.648,-122.408,-41.824,178.695,5.845,149.429
C04926=1160.643,-122.158,-41.832,178.697,5.846,149.429
C04927=1160.638,-121.908,-41.841,178.699,5.846,149.428
C04928=1160.633,-121.658,-41.850,178.701,5.846,149.428
C04929=1160.627,-121.409,-41.859,178.703,5.846,149.427
C04930=1160.622,-121.159,-41.867,178.705,5.847,149.427
C04931=1160.616,-120.908,-41.876,178.707,5.847,149.426
C04932=1160.611,-120.659,-41.884,178.709,5.848,149.426
C04933=1160.605,-120.410,-41.893,178.711,5.848,149.425
C04934=1160.601,-120.160,-41.901,178.713,5.848,149.425
C04935=1160.595,-119.910,-41.911,178.715,5.848,149.424
C04936=1160.590,-119.660,-41.920,178.717,5.849,149.424
C04937=1160.584,-119.409,-41.928,178.719,5.849,149.423
C04938=1160.578,-119.160,-41.936,178.721,5.849,149.422
C04939=1160.573,-118.910,-41.945,178.724,5.850,149.422
C04940=1160.568,-118.661,-41.954,178.725,5.850,149.421
C04941=1160.563,-118.411,-41.963,178.727,5.850,149.421
C04942=1160.557,-118.162,-41.972,178.729,5.850,149.420
C04943=1160.552,-117.912,-41.981,178.732,5.851,149.420
C04944=1160.547,-117.662,-41.989,178.733,5.851,149.419
C04945=1160.541,-117.411,-41.998,178.735,5.851,149.419
C04946=1160.536,-117.162,-42.007,178.738,5.851,149.418
C04947=1160.530,-116.912,-42.015,178.740,5.852,149.418
C04948=1160.525,-116.663,-42.024,178.741,5.852,149.417
C04949=1160.520,-116.413,-42.033,178.744,5.853,149.417
C04950=1160.515,-116.163,-42.042,178.746,5.852,149.416
C04951=1160.510,-115.913,-42.051,178.748,5.853,149.415
C04952=1160.504,-115.664,-42.059,178.749,5.853,149.415
C04953=1160.499,-115.414,-42.068,178.752,5.854,149.414
C04954=1160.493,-115.164,-42.078,178.754,5.853,149.414
C04955=1160.488,-114.914,-42.086,178.756,5.854,149.413
C04956=1160.483,-114.664,-42.095,178.758,5.855,149.413
C04957=1160.477,-114.414,-42.104,178.760,5.855,149.412
C04958=1160.472,-114.165,-42.113,178.762,5.855,149.412
C04959=1160.467,-113.915,-42.122,178.764,5.855,149.411
C04960=1160.461,-113.665,-42.131,178.766,5.856,149.411
C04961=1160.456,-113.416,-42.140,178.768,5.856,149.410
C04962=1160.451,-113.166,-42.148,178.770,5.856,149.409
C04963=1160.445,-112.916,-42.158,178.772,5.856,149.409
C04964=1160.439,-112.666,-42.166,178.774,5.857,149.408
C04965=1160.434,-112.417,-42.175,178.776,5.856,149.408
C04966=1160.429,-112.167,-42.184,178.779,5.857,149.407
C04967=1160.424,-111.917,-42.193,178.781,5.858,149.407
C04968=1160.419,-111.667,-42.202,178.782,5.858,149.406
C04969=1160.413,-111.417,-42.212,178.785,5.858,149.405
C04970=1160.408,-111.167,-42.220,178.787,5.858,149.405
C04971=1160.402,-110.917,-42.229,178.789,5.859,149.405
C04972=1160.397,-110.668,-42.238,178.790,5.859,149.404
C04973=1160.391,-110.418,-42.247,178.793,5.859,149.403
C04974=1160.386,-110.168,-42.256,178.795,5.859,149.403
C04975=1160.380,-109.918,-42.265,178.797,5.860,149.402
C04976=1160.375,-109.668,-42.274,178.800,5.860,149.402
C04977=1160.370,-109.418,-42.283,178.801,5.860,149.401
C04978=1160.365,-109.169,-42.293,178.803,5.861,149.401
C04979=1160.360,-108.919,-42.301,178.805,5.861,149.400
C04980=1160.354,-108.669,-42.311,178.808,5.861,149.399
C04981=1160.348,-108.420,-42.319,178.809,5.861,149.399
C04982=1160.343,-108.170,-42.328,178.811,5.862,149.399
C04983=1160.338,-107.920,-42.337,178.813,5.862,149.398
C04984=1160.332,-107.670,-42.347,178.816,5.863,149.397
C04985=1160.327,-107.421,-42.356,178.818,5.863,149.397
C04986=1160.322,-107.171,-42.365,178.820,5.863,149.396
C04987=1160.317,-106.921,-42.374,178.822,5.864,149.396
C04988=1160.312,-106.671,-42.383,178.824,5.864,149.395
C04989=1160.306,-106.421,-42.393,178.826,5.864,149.395
C04990=1160.301,-106.171,-42.401,178.828,5.864,149.394
C04991=1160.296,-105.922,-42.411,178.830,5.865,149.393
C04992=1160.290,-105.672,-42.421,178.832,5.866,149.393
C04993=1160.285,-105.422,-42.429,178.834,5.865,149.392
C04994=1160.280,-105.172,-42.438,178.837,5.866,149.392
C04995=1160.274,-104.922,-42.447,178.838,5.866,149.391
C04996=1160.269,-104.673,-42.457,178.841,5.866,149.391
C04997=1160.264,-104.423,-42.466,178.842,5.866,149.390
C04998=1160.258,-104.174,-42.475,178.845,5.867,149.390
C04999=1160.252,-103.924,-42.484,178.847,5.867,149.389
C05000=1160.247,-103.675,-42.494,178.849,5.867,149.388
C05001=1160.242,-103.425,-42.503,178.851,5.868,149.388
C05002=1160.237,-103.175,-42.512,178.853,5.868,149.387
C05003=1160.231,-102.925,-42.521,178.855,5.868,149.387
C05004=1160.225,-102.653,-42.532,178.858,5.869,149.386
C05005=1160.220,-102.381,-42.542,178.860,5.869,149.386
C05006=1160.214,-102.109,-42.552,178.862,5.869,149.385
C05007=1160.209,-101.837,-42.562,178.865,5.870,149.384
C05008=1160.203,-101.587,-42.572,178.866,5.870,149.384
C05009=1160.198,-101.337,-42.581,178.869,5.870,149.383
C05010=1160.193,-101.088,-42.590,178.871,5.871,149.383
C05011=1160.187,-100.838,-42.600,178.873,5.871,149.382
C05012=1160.182,-100.588,-42.609,178.875,5.871,149.381
C05013=1160.176,-100.338,-42.619,178.877,5.871,149.381
C05014=1160.171,-100.088,-42.628,178.879,5.872,149.380
C05015=1160.166,-99.838,-42.637,178.882,5.872,149.380
C05016=1160.160,-99.589,-42.647,178.883,5.872,149.379
C05017=1160.155,-99.339,-42.656,178.886,5.873,149.379
C05018=1160.149,-99.089,-42.665,178.888,5.873,149.378
C05019=1160.144,-98.840,-42.675,178.890,5.874,149.378
C05020=1160.139,-98.590,-42.684,178.892,5.874,149.377
C05021=1160.134,-98.340,-42.694,178.894,5.874,149.376
C05022=1160.129,-98.090,-42.703,178.896,5.875,149.376
C05023=1160.123,-97.840,-42.712,178.898,5.875,149.375
C05024=1160.118,-97.591,-42.722,178.901,5.875,149.375
C05025=1160.113,-97.341,-42.731,178.903,5.876,149.374
C05026=1160.107,-97.092,-42.741,178.904,5.876,149.374
C05027=1160.102,-96.842,-42.750,178.907,5.876,149.373
C05028=1160.096,-96.592,-42.760,178.909,5.876,149.373
C05029=1160.091,-96.342,-42.769,178.911,5.877,149.372
C05030=1160.085,-96.092,-42.779,178.914,5.877,149.371
C05031=1160.080,-95.843,-42.788,178.915,5.877,149.371
C05032=1160.075,-95.592,-42.798,178.917,5.878,149.370
C05033=1160.070,-95.343,-42.808,178.920,5.878,149.370
C05034=1160.064,-95.093,-42.817,178.922,5.878,149.369
C05035=1160.059,-94.844,-42.827,178.924,5.879,149.369
C05036=1160.054,-94.593,-42.836,178.926,5.879,149.368
C05037=1160.049,-94.344,-42.846,178.928,5.879,149.367
C05038=1160.043,-94.094,-42.855,178.931,5.880,149.367
C05039=1160.038,-93.845,-42.865,178.932,5.880,149.366
C05040=1160.032,-93.595,-42.874,178.935,5.881,149.366
C05041=1160.027,-93.345,-42.884,178.937,5.880,149.365
C05042=1160.021,-93.095,-42.894,178.939,5.881,149.365
C05043=1160.017,-92.845,-42.903,178.941,5.882,149.364
C05044=1160.011,-92.595,-42.913,178.943,5.881,149.363
C05045=1160.006,-92.346,-42.923,178.945,5.882,149.363
C05046=1160.001,-92.096,-42.933,178.947,5.883,149.362
C05047=1159.995,-91.846,-42.942,178.949,5.882,149.362
C05048=1159.990,-91.597,-42.952,178.952,5.883,149.361
C05049=1159.985,-91.347,-42.961,178.954,5.884,149.361
C05050=1159.979,-91.098,-42.971,178.956,5.884,149.360
C05051=1159.974,-90.847,-42.980,178.958,5.884,149.360
C05052=1159.969,-90.597,-42.990,178.960,5.884,149.359
C05053=1159.963,-90.348,-43.001,178.962,5.885,149.358
C05054=1159.958,-90.098,-43.010,178.965,5.885,149.358
C05055=1159.953,-89.848,-43.020,178.967,5.885,149.357
C05056=1159.948,-89.599,-43.029,178.969,5.886,149.357
C05057=1159.942,-89.348,-43.039,178.972,5.886,149.356
C05058=1159.938,-89.099,-43.049,178.973,5.886,149.356
C05059=1159.932,-88.849,-43.058,178.975,5.887,149.355
C05060=1159.926,-88.599,-43.069,178.978,5.887,149.354
C05061=1159.921,-88.350,-43.078,178.980,5.887,149.354
C05062=1159.915,-88.100,-43.088,178.982,5.888,149.353
C05063=1159.911,-87.850,-43.098,178.984,5.888,149.353
C05064=1159.905,-87.601,-43.108,178.986,5.888,149.352
C05065=1159.900,-87.351,-43.118,178.989,5.889,149.351
C05066=1159.895,-87.101,-43.127,178.990,5.889,149.351
C05067=1159.889,-86.852,-43.137,178.993,5.890,149.350
C05068=1159.884,-86.601,-43.148,178.995,5.890,149.350
C05069=1159.879,-86.352,-43.157,178.997,5.890,149.349
C05070=1159.873,-86.102,-43.167,178.999,5.890,149.349
C05071=1159.868,-85.852,-43.177,179.002,5.891,149.348
C05072=1159.863,-85.603,-43.187,179.003,5.891,149.348
C05073=1159.857,-85.352,-43.197,179.006,5.891,149.347
C05074=1159.853,-85.103,-43.206,179.008,5.892,149.346
C05075=1159.847,-84.854,-43.216,179.010,5.892,149.346
C05076=1159.841,-84.604,-43.227,179.012,5.893,149.345
C05077=1159.837,-84.353,-43.236,179.015,5.893,149.345
C05078=1159.831,-84.104,-43.246,179.017,5.893,149.344
C05079=1159.826,-83.854,-43.256,179.019,5.894,149.344
C05080=1159.820,-83.605,-43.266,179.021,5.895,149.343
C05081=1159.815,-83.356,-43.276,179.023,5.894,149.342
C05082=1159.810,-83.105,-43.286,179.025,5.895,149.342
C05083=1159.804,-82.855,-43.296,179.028,5.895,149.341
C05084=1159.799,-82.606,-43.306,179.030,5.895,149.341
C05085=1159.794,-82.356,-43.316,179.032,5.896,149.340
C05086=1159.789,-82.106,-43.327,179.034,5.896,149.339
C05087=1159.783,-81.856,-43.336,179.036,5.896,149.339
C05088=1159.778,-81.607,-43.346,179.039,5.897,149.338
C05089=1159.772,-81.357,-43.356,179.041,5.898,149.338
C05090=1159.767,-81.107,-43.366,179.042,5.898,149.337
C05091=1159.762,-80.857,-43.377,179.045,5.898,149.337
C05092=1159.757,-80.608,-43.386,179.047,5.899,149.336
C05093=1159.752,-80.358,-43.397,179.049,5.898,149.335
C05094=1159.746,-80.108,-43.407,179.052,5.899,149.335
C05095=1159.741,-79.858,-43.417,179.054,5.899,149.334
C05096=1159.736,-79.609,-43.426,179.057,5.900,149.334
C05097=1159.731,-79.359,-43.437,179.058,5.900,149.333
C05098=1159.725,-79.109,-43.447,179.061,5.901,149.333
C05099=1159.719,-78.860,-43.457,179.063,5.901,149.332
C05100=1159.714,-78.609,-43.468,179.065,5.901,149.331
C05101=1159.710,-78.360,-43.477,179.067,5.902,149.331
C05102=1159.704,-78.111,-43.488,179.069,5.903,149.330
C05103=1159.699,-77.860,-43.498,179.071,5.902,149.330
C05104=1159.693,-77.611,-43.508,179.074,5.903,149.329
C05105=1159.688,-77.361,-43.519,179.076,5.903,149.329
C05106=1159.683,-77.111,-43.529,179.078,5.903,149.328
C05107=1159.678,-76.862,-43.539,179.080,5.904,149.328
C05108=1159.671,-76.591,-43.550,179.083,5.904,149.327
C05109=1159.666,-76.320,-43.561,179.085,5.905,149.326
C05110=1159.660,-76.048,-43.572,179.088,5.906,149.326
C05111=1159.654,-75.776,-43.584,179.090,5.906,149.325
C05112=1159.650,-75.527,-43.594,179.092,5.906,149.324
C05113=1159.644,-75.278,-43.604,179.095,5.906,149.324
C05114=1159.639,-75.027,-43.614,179.097,5.907,149.323
C05115=1159.633,-74.778,-43.625,179.099,5.907,149.323
C05116=1159.628,-74.528,-43.635,179.101,5.908,149.322
C05117=1159.623,-74.278,-43.645,179.104,5.908,149.321
C05118=1159.617,-74.029,-43.656,179.105,5.908,149.321
C05119=1159.612,-73.779,-43.666,179.108,5.909,149.320
C05120=1159.607,-73.529,-43.676,179.110,5.909,149.320
C05121=1159.602,-73.280,-43.686,179.112,5.910,149.319
C05122=1159.596,-73.030,-43.696,179.114,5.909,149.319
C05123=1159.591,-72.780,-43.707,179.117,5.910,149.318
C05124=1159.586,-72.530,-43.717,179.119,5.911,149.317
C05125=1159.581,-72.281,-43.728,179.121,5.911,149.317
C05126=1159.575,-72.031,-43.738,179.123,5.911,149.316
C05127=1159.570,-71.782,-43.749,179.126,5.912,149.316
C05128=1159.565,-71.531,-43.759,179.128,5.913,149.315
C05129=1159.559,-71.282,-43.769,179.130,5.912,149.314
C05130=1159.554,-71.031,-43.780,179.132,5.913,149.314
C05131=1159.548,-70.782,-43.790,179.135,5.913,149.313
C05132=1159.543,-70.533,-43.801,179.137,5.914,149.313
C05133=1159.538,-70.283,-43.812,179.139,5.914,149.312
C05134=1159.533,-70.033,-43.822,179.141,5.914,149.312
C05135=1159.528,-69.783,-43.832,179.144,5.915,149.311
C05136=1159.522,-69.533,-43.843,179.146,5.915,149.310
C05137=1159.517,-69.283,-43.853,179.148,5.916,149.310
C05138=1159.512,-69.034,-43.864,179.150,5.916,149.309
C05139=1159.506,-68.785,-43.874,179.153,5.917,149.309
C05140=1159.501,-68.534,-43.885,179.155,5.916,149.308
C05141=1159.495,-68.285,-43.895,179.157,5.917,149.308
C05142=1159.490,-68.035,-43.906,179.160,5.918,149.307
C05143=1159.485,-67.786,-43.917,179.162,5.918,149.306
C05144=1159.480,-67.536,-43.927,179.163,5.918,149.306
C05145=1159.475,-67.286,-43.937,179.166,5.919,149.305
C05146=1159.470,-67.036,-43.948,179.168,5.920,149.305
C05147=1159.464,-66.787,-43.959,179.171,5.920,149.304
C05148=1159.459,-66.537,-43.970,179.172,5.920,149.304
C05149=1159.454,-66.287,-43.980,179.175,5.920,149.303
C05150=1159.448,-66.038,-43.991,179.177,5.921,149.302
C05151=1159.443,-65.788,-44.001,179.180,5.922,149.302
C05152=1159.438,-65.538,-44.011,179.182,5.922,149.301
C05153=1159.433,-65.289,-44.023,179.184,5.922,149.301
C05154=1159.428,-65.039,-44.033,179.186,5.923,149.300
C05155=1159.422,-64.789,-44.044,179.189,5.923,149.299
C05156=1159.416,-64.539,-44.054,179.191,5.923,149.299
C05157=1159.411,-64.289,-44.066,179.193,5.924,149.298
C05158=1159.406,-64.040,-44.076,179.196,5.924,149.298
C05159=1159.401,-63.790,-44.087,179.198,5.925,149.297
C05160=1159.396,-63.541,-44.097,179.200,5.925,149.296
C05161=1159.391,-63.290,-44.108,179.202,5.925,149.296
C05162=1159.386,-63.041,-44.119,179.205,5.926,149.295
C05163=1159.380,-62.791,-44.129,179.207,5.927,149.295
C05164=1159.375,-62.541,-44.140,179.209,5.926,149.294
C05165=1159.369,-62.292,-44.151,179.211,5.927,149.294
C05166=1159.364,-62.042,-44.162,179.213,5.928,149.293
C05167=1159.359,-61.793,-44.173,179.216,5.928,149.292
C05168=1159.354,-61.542,-44.184,179.218,5.929,149.292
C05169=1159.348,-61.293,-44.194,179.220,5.929,149.291
C05170=1159.344,-61.043,-44.205,179.222,5.929,149.291
C05171=1159.337,-60.793,-44.216,179.225,5.930,149.290
C05172=1159.333,-60.544,-44.227,179.227,5.931,149.290
C05173=1159.328,-60.294,-44.238,179.229,5.930,149.289
C05174=1159.322,-60.045,-44.249,179.232,5.931,149.288
C05175=1159.317,-59.794,-44.259,179.234,5.931,149.288
C05176=1159.312,-59.545,-44.270,179.236,5.932,149.287
C05177=1159.306,-59.295,-44.281,179.239,5.932,149.286
C05178=1159.301,-59.046,-44.292,179.241,5.933,149.286
C05179=1159.296,-58.796,-44.303,179.243,5.933,149.285
C05180=1159.291,-58.546,-44.314,179.246,5.934,149.285
C05181=1159.286,-58.297,-44.324,179.248,5.935,149.284
C05182=1159.280,-58.047,-44.336,179.250,5.934,149.284
C05183=1159.275,-57.797,-44.346,179.252,5.935,149.283
C05184=1159.270,-57.547,-44.358,179.255,5.935,149.282
C05185=1159.265,-57.297,-44.368,179.257,5.936,149.282
C05186=1159.259,-57.048,-44.380,179.260,5.936,149.281
C05187=1159.254,-56.798,-44.390,179.261,5.937,149.281
C05188=1159.249,-56.549,-44.401,179.264,5.937,149.280
C05189=1159.244,-56.299,-44.413,179.266,5.938,149.280
C05190=1159.238,-56.049,-44.424,179.269,5.938,149.279
C05191=1159.233,-55.800,-44.435,179.271,5.939,149.278
C05192=1159.228,-55.549,-44.445,179.273,5.938,149.278
C05193=1159.223,-55.300,-44.457,179.275,5.939,149.277
C05194=1159.217,-55.051,-44.468,179.278,5.940,149.277
C05195=1159.212,-54.800,-44.479,179.280,5.940,149.276
C05196=1159.208,-54.551,-44.490,179.283,5.941,149.275
C05197=1159.202,-54.301,-44.500,179.284,5.941,149.275
C05198=1159.197,-54.051,-44.512,179.287,5.941,149.274
C05199=1159.192,-53.802,-44.523,179.289,5.942,149.274
C05200=1159.186,-53.552,-44.534,179.292,5.942,149.273
C05201=1159.181,-53.302,-44.545,179.294,5.943,149.272
C05202=1159.176,-53.052,-44.557,179.296,5.943,149.272
C05203=1159.171,-52.803,-44.567,179.298,5.944,149.271
C05204=1159.165,-52.553,-44.579,179.301,5.944,149.271
C05205=1159.160,-52.303,-44.590,179.303,5.945,149.270
C05206=1159.155,-52.054,-44.601,179.305,5.946,149.270
C05207=1159.149,-51.804,-44.612,179.308,5.946,149.269
C05208=1159.145,-51.554,-44.623,179.309,5.946,149.268
C05209=1159.139,-51.305,-44.634,179.312,5.946,149.268
C05210=1159.134,-51.055,-44.646,179.314,5.947,149.267
C05211=1159.129,-50.805,-44.657,179.317,5.948,149.267
C05212=1159.123,-50.535,-44.669,179.320,5.948,149.266
C05213=1159.117,-50.265,-44.682,179.322,5.949,149.265
C05214=1159.112,-49.994,-44.694,179.325,5.949,149.265
C05215=1159.106,-49.723,-44.706,179.327,5.950,149.264
C05216=1159.101,-49.474,-44.717,179.329,5.950,149.264
C05217=1159.096,-49.224,-44.729,179.331,5.950,149.263
C05218=1159.090,-48.974,-44.739,179.334,5.951,149.262
C05219=1159.085,-48.725,-44.750,179.336,5.951,149.262
C05220=1159.080,-48.475,-44.762,179.338,5.952,149.261
C05221=1159.075,-48.226,-44.773,179.341,5.952,149.260
C05222=1159.069,-47.976,-44.785,179.343,5.953,149.260
C05223=1159.064,-47.725,-44.796,179.345,5.953,149.259
C05224=1159.059,-47.476,-44.808,179.348,5.954,149.259
C05225=1159.053,-47.227,-44.819,179.350,5.954,149.258
C05226=1159.048,-46.977,-44.830,179.352,5.955,149.258
C05227=1159.043,-46.727,-44.842,179.355,5.955,149.257
C05228=1159.039,-46.477,-44.853,179.357,5.956,149.256
C05229=1159.033,-46.228,-44.865,179.359,5.956,149.256
C05230=1159.028,-45.978,-44.875,179.362,5.956,149.255
C05231=1159.022,-45.728,-44.887,179.364,5.957,149.255
C05232=1159.017,-45.478,-44.898,179.366,5.958,149.254
C05233=1159.012,-45.228,-44.910,179.369,5.958,149.253
C05234=1159.007,-44.980,-44.921,179.371,5.959,149.253
C05235=1159.001,-44.730,-44.933,179.374,5.959,149.252
C05236=1158.997,-44.480,-44.944,179.376,5.959,149.252
C05237=1158.991,-44.230,-44.956,179.378,5.960,149.251
C05238=1158.986,-43.981,-44.967,179.380,5.961,149.251
C05239=1158.980,-43.731,-44.979,179.383,5.961,149.250
C05240=1158.975,-43.481,-44.991,179.385,5.962,149.249
C05241=1158.970,-43.232,-45.002,179.388,5.962,149.249
C05242=1158.965,-42.982,-45.014,179.390,5.963,149.248
C05243=1158.960,-42.732,-45.025,179.392,5.963,149.248
C05244=1158.954,-42.483,-45.037,179.394,5.963,149.247
C05245=1158.949,-42.233,-45.048,179.397,5.964,149.246
C05246=1158.944,-41.983,-45.060,179.399,5.965,149.246
C05247=1158.939,-41.734,-45.071,179.402,5.965,149.245
C05248=1158.934,-41.484,-45.083,179.404,5.966,149.245
C05249=1158.928,-41.234,-45.095,179.407,5.966,149.244
C05250=1158.923,-40.985,-45.106,179.409,5.967,149.244
C05251=1158.918,-40.735,-45.118,179.411,5.967,149.243
C05252=1158.913,-40.485,-45.129,179.413,5.967,149.242
C05253=1158.908,-40.235,-45.141,179.416,5.968,149.242
C05254=1158.902,-39.985,-45.153,179.418,5.969,149.241
C05255=1158.898,-39.736,-45.164,179.421,5.969,149.240
C05256=1158.891,-39.487,-45.176,179.423,5.970,149.240
C05257=1158.886,-39.237,-45.188,179.425,5.970,149.239
C05258=1158.881,-38.987,-45.199,179.428,5.971,149.239
C05259=1158.876,-38.737,-45.211,179.430,5.971,149.238
C05260=1158.871,-38.487,-45.222,179.432,5.971,149.238
C05261=1158.866,-38.238,-45.235,179.435,5.972,149.237
C05262=1158.861,-37.988,-45.247,179.437,5.973,149.236
C05263=1158.856,-37.739,-45.258,179.439,5.973,149.236
C05264=1158.850,-37.489,-45.269,179.442,5.974,149.235
C05265=1158.845,-37.239,-45.281,179.444,5.974,149.235
C05266=1158.839,-36.989,-45.293,179.446,5.975,149.234
C05267=1158.834,-36.740,-45.304,179.449,5.976,149.233
C05268=1158.829,-36.490,-45.317,179.451,5.976,149.233
C05269=1158.824,-36.241,-45.329,179.453,5.976,149.232
C05270=1158.819,-35.991,-45.340,179.456,5.977,149.232
C05271=1158.814,-35.741,-45.352,179.458,5.977,149.231
C05272=1158.808,-35.491,-45.364,179.460,5.978,149.231
C05273=1158.804,-35.242,-45.376,179.463,5.978,149.230
C05274=1158.798,-34.993,-45.388,179.465,5.979,149.229
C05275=1158.792,-34.743,-45.399,179.468,5.980,149.229
C05276=1158.787,-34.493,-45.411,179.470,5.980,149.228
C05277=1158.782,-34.243,-45.423,179.473,5.981,149.228
C05278=1158.777,-33.994,-45.435,179.475,5.982,149.227
C05279=1158.772,-33.744,-45.447,179.477,5.981,149.226
C05280=1158.766,-33.494,-45.459,179.479,5.982,149.226
C05281=1158.762,-33.245,-45.471,179.482,5.982,149.225
C05282=1158.757,-32.995,-45.483,179.484,5.983,149.225
C05283=1158.751,-32.745,-45.495,179.487,5.984,149.224
C05284=1158.746,-32.495,-45.507,179.489,5.984,149.223
C05285=1158.741,-32.246,-45.519,179.492,5.985,149.223
C05286=1158.736,-31.996,-45.531,179.494,5.985,149.222
C05287=1158.730,-31.746,-45.542,179.496,5.986,149.222
C05288=1158.725,-31.497,-45.555,179.499,5.987,149.221
C05289=1158.720,-31.247,-45.567,179.501,5.987,149.221
C05290=1158.714,-30.997,-45.579,179.504,5.988,149.220
C05291=1158.710,-30.748,-45.591,179.506,5.989,149.219
C05292=1158.705,-30.498,-45.603,179.508,5.988,149.219
C05293=1158.699,-30.248,-45.615,179.510,5.989,149.218
C05294=1158.694,-29.999,-45.627,179.513,5.989,149.217
C05295=1158.689,-29.749,-45.639,179.515,5.990,149.217
C05296=1158.684,-29.500,-45.652,179.518,5.991,149.216
C05297=1158.679,-29.250,-45.663,179.520,5.991,149.216
C05298=1158.673,-29.000,-45.675,179.523,5.992,149.215
C05299=1158.668,-28.751,-45.687,179.525,5.993,149.215
C05300=1158.663,-28.501,-45.699,179.528,5.993,149.214
C05301=1158.658,-28.252,-45.712,179.530,5.994,149.214
C05302=1158.652,-28.002,-45.724,179.532,5.994,149.213
C05303=1158.647,-27.752,-45.736,179.535,5.995,149.212
C05304=1158.642,-27.502,-45.748,179.537,5.996,149.212
C05305=1158.637,-27.253,-45.760,179.539,5.996,149.211
C05306=1158.632,-27.004,-45.772,179.542,5.997,149.210
C05307=1158.626,-26.754,-45.784,179.544,5.998,149.210
C05308=1158.621,-26.504,-45.797,179.547,5.998,149.209
C05309=1158.616,-26.254,-45.809,179.550,5.998,149.209
C05310=1158.611,-26.005,-45.821,179.551,5.998,149.208
C05311=1158.606,-25.754,-45.833,179.554,5.999,149.207
C05312=1158.601,-25.505,-45.846,179.556,6.000,149.207
C05313=1158.596,-25.256,-45.859,179.559,6.000,149.206
C05314=1158.590,-25.006,-45.870,179.561,6.001,149.206
C05315=1158.585,-24.756,-45.883,179.563,6.001,149.205
C05316=1158.580,-24.486,-45.896,179.566,6.002,149.205
C05317=1158.574,-24.216,-45.909,179.568,6.003,149.204
C05318=1158.569,-23.947,-45.922,179.572,6.004,149.203
C05319=1158.562,-23.677,-45.936,179.574,6.004,149.203
C05320=1158.558,-23.427,-45.948,179.576,6.005,149.202
C05321=1158.552,-23.177,-45.960,179.579,6.005,149.201
C05322=1158.547,-22.928,-45.973,179.581,6.006,149.201
C05323=1158.542,-22.678,-45.986,179.584,6.007,149.200
C05324=1158.537,-22.428,-45.997,179.586,6.008,149.200
C05325=1158.532,-22.179,-46.010,179.589,6.008,149.199
C05326=1158.526,-21.930,-46.023,179.591,6.009,149.199
C05327=1158.521,-21.680,-46.035,179.594,6.009,149.198
C05328=1158.516,-21.430,-46.047,179.596,6.010,149.197
C05329=1158.511,-21.180,-46.060,179.598,6.010,149.197
C05330=1158.506,-20.930,-46.072,179.600,6.010,149.196
C05331=1158.501,-20.681,-46.085,179.603,6.011,149.196
C05332=1158.496,-20.432,-46.097,179.605,6.012,149.195
C05333=1158.490,-20.182,-46.109,179.608,6.012,149.194
C05334=1158.485,-19.933,-46.122,179.610,6.013,149.194
C05335=1158.480,-19.683,-46.134,179.612,6.013,149.193
C05336=1158.475,-19.433,-46.147,179.615,6.014,149.193
C05337=1158.470,-19.183,-46.159,179.617,6.015,149.192
C05338=1158.464,-18.934,-46.172,179.620,6.015,149.191
C05339=1158.459,-18.684,-46.185,179.622,6.016,149.191
C05340=1158.454,-18.434,-46.197,179.625,6.016,149.190
C05341=1158.449,-18.185,-46.209,179.627,6.017,149.190
C05342=1158.444,-17.935,-46.222,179.630,6.018,149.189
C05343=1158.439,-17.686,-46.235,179.632,6.018,149.189
C05344=1158.433,-17.436,-46.247,179.634,6.019,149.188
C05345=1158.428,-17.186,-46.259,179.637,6.020,149.187
C05346=1158.423,-16.937,-46.272,179.639,6.020,149.187
C05347=1158.418,-16.687,-46.286,179.641,6.021,149.186
C05348=1158.413,-16.438,-46.298,179.644,6.021,149.186
C05349=1158.407,-16.188,-46.310,179.646,6.022,149.185
C05350=1158.402,-15.938,-46.323,179.649,6.022,149.184
C05351=1158.398,-15.688,-46.336,179.651,6.023,149.184
C05352=1158.393,-15.439,-46.348,179.654,6.024,149.183
C05353=1158.387,-15.189,-46.361,179.656,6.025,149.183
C05354=1158.382,-14.940,-46.374,179.659,6.026,149.182
C05355=1158.376,-14.690,-46.386,179.662,6.026,149.181
C05356=1158.372,-14.440,-46.399,179.664,6.027,149.181
C05357=1158.367,-14.191,-46.412,179.667,6.027,149.180
C05358=1158.361,-13.941,-46.424,179.669,6.028,149.180
C05359=1158.356,-13.692,-46.437,179.672,6.029,149.179
C05360=1158.351,-13.442,-46.450,179.674,6.030,149.179
C05361=1158.346,-13.192,-46.463,179.676,6.030,149.178
C05362=1158.341,-12.943,-46.476,179.679,6.031,149.177
C05363=1158.336,-12.693,-46.489,179.681,6.031,149.177
C05364=1158.330,-12.443,-46.502,179.683,6.032,149.176
C05365=1158.325,-12.194,-46.514,179.686,6.032,149.176
C05366=1158.320,-11.945,-46.527,179.688,6.033,149.175
C05367=1158.315,-11.694,-46.540,179.691,6.034,149.174
C05368=1158.309,-11.445,-46.552,179.693,6.035,149.174
C05369=1158.304,-11.195,-46.565,179.696,6.035,149.173
C05370=1158.300,-10.945,-46.578,179.698,6.036,149.173
C05371=1158.294,-10.696,-46.591,179.701,6.036,149.172
C05372=1158.289,-10.446,-46.604,179.703,6.037,149.171
C05373=1158.284,-10.197,-46.616,179.705,6.037,149.171
C05374=1158.280,-9.948,-46.630,179.708,6.038,149.170
C05375=1158.274,-9.698,-46.643,179.710,6.039,149.170
C05376=1158.269,-9.449,-46.656,179.713,6.039,149.169
C05377=1158.264,-9.199,-46.669,179.715,6.040,149.169
C05378=1158.258,-8.949,-46.682,179.718,6.040,149.168
C05379=1158.253,-8.700,-46.695,179.720,6.041,149.167
C05380=1158.248,-8.450,-46.707,179.723,6.042,149.167
C05381=1158.243,-8.200,-46.721,179.725,6.043,149.166
C05382=1158.238,-7.951,-46.733,179.728,6.044,149.166
C05383=1158.233,-7.701,-46.746,179.730,6.045,149.165
C05384=1158.227,-7.451,-46.759,179.733,6.045,149.164
C05385=1158.223,-7.201,-46.772,179.735,6.046,149.164
C05386=1158.217,-6.952,-46.785,179.738,6.046,149.163
C05387=1158.212,-6.703,-46.799,179.740,6.047,149.163
C05388=1158.207,-6.453,-46.812,179.742,6.048,149.162
C05389=1158.202,-6.203,-46.825,179.745,6.048,149.161
C05390=1158.196,-5.954,-46.838,179.747,6.049,149.161
C05391=1158.192,-5.704,-46.851,179.750,6.049,149.160
C05392=1158.186,-5.454,-46.864,179.752,6.050,149.160
C05393=1158.181,-5.205,-46.877,179.755,6.050,149.159
C05394=1158.176,-4.955,-46.891,179.757,6.051,149.159
C05395=1158.171,-4.706,-46.903,179.760,6.052,149.158
C05396=1158.166,-4.456,-46.916,179.762,6.053,149.157
C05397=1158.160,-4.206,-46.929,179.765,6.054,149.157
C05398=1158.156,-3.957,-46.943,179.767,6.055,149.156
C05399=1158.150,-3.707,-46.956,179.770,6.055,149.156
C05400=1158.145,-3.458,-46.969,179.772,6.056,149.155
C05401=1158.140,-3.207,-46.983,179.775,6.056,149.154
C05402=1158.135,-2.959,-46.996,179.777,6.057,149.154
C05403=1158.130,-2.708,-47.009,179.780,6.058,149.153
C05404=1158.125,-2.459,-47.022,179.782,6.058,149.153
C05405=1158.120,-2.210,-47.035,179.784,6.059,149.152
C05406=1158.115,-1.960,-47.049,179.787,6.059,149.152
C05407=1158.110,-1.711,-47.061,179.789,6.060,149.151
C05408=1158.104,-1.460,-47.075,179.792,6.061,149.150
C05409=1158.099,-1.212,-47.088,179.795,6.062,149.150
C05410=1158.094,-0.961,-47.102,179.797,6.063,149.149
C05411=1158.088,-0.712,-47.115,179.799,6.063,149.149
C05412=1158.084,-0.462,-47.129,179.802,6.064,149.148
C05413=1158.078,-0.213,-47.142,179.804,6.065,149.148
C05414=1158.074,0.037,-47.155,179.807,6.065,149.147
C05415=1158.068,0.286,-47.169,179.809,6.066,149.146
C05416=1158.063,0.536,-47.181,179.812,6.066,149.146
C05417=1158.058,0.786,-47.195,179.815,6.068,149.145
C05418=1158.053,1.035,-47.208,179.817,6.068,149.145
C05419=1158.048,1.285,-47.222,179.819,6.069,149.144
C05420=1158.042,1.554,-47.237,179.822,6.070,149.143
C05421=1158.037,1.823,-47.251,179.825,6.070,149.143
C05422=1158.031,2.093,-47.265,179.828,6.071,149.142
C05423=1158.026,2.362,-47.280,179.830,6.072,149.142
C05424=1158.021,2.612,-47.293,179.833,6.073,149.141
C05425=1158.016,2.861,-47.307,179.835,6.074,149.140
C05426=1158.010,3.111,-47.320,179.838,6.074,149.140
C05427=1158.006,3.360,-47.334,179.840,6.075,149.139
C05428=1158.000,3.610,-47.347,179.842,6.075,149.139
C05429=1157.995,3.860,-47.361,179.845,6.077,149.138
C05430=1157.990,4.109,-47.374,179.848,6.077,149.137
C05431=1157.985,4.359,-47.388,179.850,6.078,149.137
C05432=1157.980,4.609,-47.401,179.853,6.079,149.136
C05433=1157.975,4.858,-47.415,179.855,6.079,149.136
C05434=1157.969,5.108,-47.429,179.857,6.080,149.135
C05435=1157.965,5.357,-47.442,179.860,6.080,149.134
C05436=1157.959,5.607,-47.456,179.863,6.082,149.134
C05437=1157.954,5.856,-47.470,179.866,6.082,149.133
C05438=1157.949,6.106,-47.483,179.868,6.083,149.133
C05439=1157.944,6.356,-47.497,179.870,6.084,149.132
C05440=1157.939,6.605,-47.511,179.873,6.085,149.132
C05441=1157.934,6.855,-47.524,179.875,6.085,149.131
C05442=1157.929,7.104,-47.538,179.877,6.086,149.131
C05443=1157.923,7.354,-47.551,179.881,6.087,149.130
C05444=1157.918,7.603,-47.565,179.883,6.088,149.129
C05445=1157.914,7.853,-47.579,179.885,6.088,149.129
C05446=1157.908,8.103,-47.592,179.888,6.089,149.128
C05447=1157.903,8.352,-47.606,179.890,6.090,149.128
C05448=1157.899,8.601,-47.620,179.892,6.090,149.127
C05449=1157.893,8.851,-47.633,179.895,6.091,149.126
C05450=1157.888,9.101,-47.647,179.898,6.093,149.126
C05451=1157.883,9.350,-47.662,179.900,6.093,149.125
C05452=1157.878,9.600,-47.674,179.903,6.094,149.125
C05453=1157.873,9.849,-47.689,179.905,6.094,149.124
C05454=1157.868,10.099,-47.703,179.907,6.095,149.124
C05455=1157.862,10.349,-47.716,179.910,6.096,149.123
C05456=1157.857,10.598,-47.730,179.913,6.097,149.122
C05457=1157.852,10.847,-47.744,179.916,6.098,149.122
C05458=1157.847,11.097,-47.758,179.918,6.098,149.121
C05459=1157.842,11.347,-47.771,179.920,6.099,149.121
C05460=1157.836,11.596,-47.785,179.923,6.099,149.120
C05461=1157.831,11.846,-47.800,179.925,6.100,149.120
C05462=1157.827,12.095,-47.813,179.928,6.101,149.119
C05463=1157.821,12.345,-47.826,179.931,6.102,149.118
C05464=1157.816,12.595,-47.841,179.933,6.103,149.118
C05465=1157.811,12.844,-47.855,179.935,6.104,149.117
C05466=1157.806,13.093,-47.869,179.938,6.104,149.117
C05467=1157.801,13.343,-47.883,179.941,6.106,149.116
C05468=1157.796,13.593,-47.897,179.943,6.106,149.115
C05469=1157.792,13.843,-47.910,179.946,6.107,149.115
C05470=1157.786,14.092,-47.924,179.948,6.107,149.114
C05471=1157.781,14.342,-47.939,179.950,6.108,149.114
C05472=1157.776,14.591,-47.953,179.953,6.109,149.113
C05473=1157.770,14.840,-47.967,179.956,6.110,149.113
C05474=1157.765,15.091,-47.980,179.959,6.111,149.112
C05475=1157.760,15.340,-47.995,179.961,6.112,149.112
C05476=1157.755,15.589,-48.009,179.963,6.112,149.111
C05477=1157.750,15.839,-48.023,179.966,6.113,149.110
C05478=1157.746,16.088,-48.037,179.969,6.114,149.110
C05479=1157.741,16.338,-48.051,179.971,6.115,149.109
C05480=1157.735,16.587,-48.065,179.974,6.115,149.109
C05481=1157.730,16.837,-48.079,179.976,6.116,149.108
C05482=1157.725,17.087,-48.093,179.978,6.117,149.107
C05483=1157.720,17.336,-48.108,179.981,6.118,149.107
C05484=1157.715,17.585,-48.121,179.984,6.119,149.106
C05485=1157.710,17.835,-48.136,179.986,6.120,149.106
C05486=1157.705,18.085,-48.150,179.989,6.120,149.105
C05487=1157.700,18.334,-48.164,179.991,6.122,149.105
C05488=1157.694,18.583,-48.178,179.994,6.122,149.104
C05489=1157.689,18.833,-48.193,179.996,6.123,149.104
C05490=1157.684,19.083,-48.207,179.999,6.124,149.103
C05491=1157.679,19.333,-48.221,-179.998,6.124,149.102
C05492=1157.674,19.582,-48.235,-179.996,6.126,149.102
C05493=1157.669,19.831,-48.249,-179.993,6.126,149.101
C05494=1157.664,20.081,-48.264,-179.991,6.127,149.101
C05495=1157.659,20.331,-48.278,-179.988,6.127,149.100
C05496=1157.654,20.580,-48.292,-179.985,6.129,149.100
C05497=1157.649,20.830,-48.306,-179.983,6.129,149.099
C05498=1157.643,21.079,-48.320,-179.981,6.130,149.098
C05499=1157.638,21.329,-48.335,-179.978,6.131,149.098
C05500=1157.634,21.579,-48.349,-179.976,6.132,149.097
